// TIA Portal project "ManufacturingCell2_ATOLE" (V19)

(* hardware
DEVICE "S7-1200 station_1"  S7-1200 Station
   slot 0: "Rack_0"  S7-1200 Rack  Rack  V1.0
   slot 1: "PLC_Machining"  CPU 1214C AC/DC/Rly  6ES7 214-1BG40-0XB0  V4.5
   slot 2: "DI 16x24VDC/DQ 16xRelay_1"  SM 1223 DI16/DQ16 x relay  6ES7 223-1PL32-0XB0  V2.0
   slot 3: "AQ 1x12BIT_1"  AQ1 signal board  6ES7 232-4HA30-0XB0  V1.0
   slot 3: "AI 4x13BIT/AQ 2x14BIT_1"  6ES7 234-4HE32-0XB0  V2.1
DEVICE "Machining_HMI"  KTP700 Basic PN
   slot 0: "HMI_1"  KTP700 Basic PN  6AV2 123-2GB03-0AX0  17.0.0.0
   slot 1: "HMI_RT_1"  KTP700 Basic PN  6AV2 123-2GB03-0AX0  17.0.0.0
   slot 5: "HMI_1.IE_CP_1"  PROFINET Interface  17.0.0.0
      slot 1: "PROFINET Interface_1"  PROFINET Interface
         slot 1: "Port_1"  Port
DEVICE "S7-1200 station_2"  S7-1200 Station
   slot 0: "Rack_0"  S7-1200 Rack  Rack  V1.0
   slot 1: "PLC_Pneumatic"  CPU 1214C AC/DC/Rly  6ES7 214-1BG40-0XB0  V4.5
   slot 2: "DI 16x24VDC/DQ 16xRelay_1"  SM 1223 DI16/DQ16 x relay  6ES7 223-1PL32-0XB0  V2.0
   slot 3: "AQ 1x12BIT_1"  AQ1 signal board  6ES7 232-4HA30-0XB0  V1.0
   slot 3: "AI 4x13BIT/AQ 2x14BIT_1"  6ES7 234-4HE32-0XB0  V2.1
DEVICE "Pneumatic_HMI"  KTP700 Basic PN
   slot 0: "HMI_2"  KTP700 Basic PN  6AV2 123-2GB03-0AX0  17.0.0.0
   slot 1: "HMI_RT_2"  KTP700 Basic PN  6AV2 123-2GB03-0AX0  17.0.0.0
   slot 5: "HMI_2.IE_CP_1"  PROFINET Interface  17.0.0.0
      slot 1: "PROFINET Interface_1"  PROFINET Interface
         slot 1: "Port_1"  Port
*)

// ===== PLC "PLC_Machining"  CPU 1214C AC/DC/Rly =====

VAR_GLOBAL   // PLC tag table "Default tag table"
   "Pusher_latch" AT %M10.0 : Bool;
   "Conveyor2_latch" AT %M10.1 : Bool;
   "Conveyor4_latch" AT %M10.2 : Bool;
   "Conveyor3_latch" AT %M10.3 : Bool;
   "Conveyor5_latch" AT %M10.4 : Bool;
   "Conveyor6_IN_latch" AT %M10.5 : Bool;
   "Conveyor6_OUT_latch" AT %M10.6 : Bool;
   "Conveyor6_Position" AT %M10.7 : Bool;
   "lampBlinkTag" AT %M11.0 : Bool;
   "cakeFlavor" AT %MW12 : UInt;
   "drillingTime" AT %MD14 : Time;
   "mixingTime" AT %MD18 : Time;
   "System_Byte" AT %MB22 : Byte;
   "FirstScan" AT %M22.0 : Bool;
   "DiagStatusUpdate" AT %M22.1 : Bool;
   "AlwaysTRUE" AT %M22.2 : Bool;
   "AlwaysFALSE" AT %M22.3 : Bool;
   "drillActive" AT %M23.0 : Bool;
   "mixActive" AT %M23.1 : Bool;
   "CognexID" AT %MW24 : Int;
   "manualModeSW_memory" AT %M23.2 : Bool;
   "CognexID_UInt" AT %MW26 : UInt;
   "SetCognexID_Edge" AT %M23.3 : Bool;
   "OptoDrill_Edge" AT %M23.4 : Bool;
   "OptoMix_Edge" AT %M23.5 : Bool;
   "Power_consumption" AT %MD28 : Real;
   "Conveyor6_OUT_Finish" AT %M11.1 : Bool;
   "Conveyor6Finish_TP_Edge" AT %M11.2 : Bool;
END_VAR

VAR_GLOBAL   // PLC tag table "M_HMI_Tags"
   "HMI_BTN_Conveyor2" AT %M50.1 : Bool;
   "HMI_BTN_Pusher1" AT %M50.2 : Bool;
   "HMI_BTN_Conveyor3" AT %M50.3 : Bool;
   "HMI_BTN_Conveyor4" AT %M50.4 : Bool;
   "HMI_BTN_Conveyor5" AT %M50.5 : Bool;
   "HMI_BTN_Drill" AT %M50.6 : Bool;
   "HMI_BTN_Mix" AT %M50.7 : Bool;
   "HMI_BTN1" AT %M50.0 : Bool;
   "HMI_BTN_Pusher2" AT %M51.0 : Bool;
   "HMI_BTN_Conveyor6IN" AT %M51.1 : Bool;
   "HMI_BTN_Conveyor6OUT" AT %M51.2 : Bool;
   "HMI_BTN_PressDown" AT %M51.3 : Bool;
   "HMI_BTN_PressUp" AT %M51.4 : Bool;
   "HMI_BTN_PlantView" AT %M51.5 : Bool;
   "HMI_BTN_ProcessTimes" AT %M51.6 : Bool;
   "HMI_BTN_ManualControl" AT %M51.7 : Bool;
   "HMI_BTN17" AT %M52.0 : Bool;
   "HMI_BTN18" AT %M52.1 : Bool;
   "HMI_BTN19" AT %M52.2 : Bool;
   "HMI_BTN20" AT %M52.3 : Bool;
   "HMI_BTN21" AT %M52.4 : Bool;
   "HMI_BTN22" AT %M52.5 : Bool;
   "HMI_BTN23" AT %M52.6 : Bool;
   "HMI_BTN24" AT %M52.7 : Bool;
   "ManualMode_SW" AT %M53.0 : Bool;
   "HMI_SetScreen" AT %MW54 : Int;
END_VAR

VAR_GLOBAL   // PLC tag table "M_Cell_Tags"
   "Opto_Conveyor2A" AT %I0.0 : Bool;
   "Opto_Conveyor2B" AT %I0.1 : Bool;
   "Green_BTN" AT %I9.4 : Bool;
   "Yellow_BTN" AT %I9.5 : Bool;
   "Red_BTN" AT %I9.6 : Bool;
   "Emergency_BTN" AT %I9.7 : Bool;
   "Pusher1_BTN" AT %I0.2 : Bool;
   "Opto_Drill" AT %I0.3 : Bool;
   "Opto_Mix" AT %I0.4 : Bool;
   "Opto_Conveyor5" AT %I0.6 : Bool;
   "Pusher2_BTN" AT %I0.5 : Bool;
   "Opto_Conveyor6A" AT %I8.1 : Bool;
   "Opto_Conveyor6B" AT %I8.0 : Bool;
   "Press_BTN_DOWN" AT %I8.2 : Bool;
   "Press_BTN_UP" AT %I8.3 : Bool;
   "Conveyor2_tactileSW" AT %I0.7 : Bool;
   "cellPotentiometer" AT %IW64 : Int;
   "Cognex_out0" AT %I9.0 : Bool;
   "Cognex_out1" AT %I9.1 : Bool;
   "Cognex_out2" AT %I9.2 : Bool;
   "Green_Light" AT %Q9.5 : Bool;
   "Red_Light" AT %Q9.6 : Bool;
   "Blue_Light" AT %Q9.7 : Bool;
   "Conveyor2" AT %Q0.0 : Bool;
   "Pusher1" AT %Q0.1 : Bool;
   "Conveyor4" AT %Q0.4 : Bool;
   "Conveyor5" AT %Q0.7 : Bool;
   "Conveyor3" AT %Q0.2 : Bool;
   "Drill" AT %Q0.3 : Bool;
   "Mix" AT %Q0.5 : Bool;
   "Pusher2" AT %Q0.6 : Bool;
   "Green_Tower" AT %Q1.0 : Bool;
   "Red_Tower" AT %Q1.1 : Bool;
   "Conveyor6_OUT" AT %Q8.3 : Bool;
   "Press_UP" AT %Q8.4 : Bool;
   "Press_DOWN" AT %Q8.5 : Bool;
   "Conveyor6_IN" AT %Q8.2 : Bool;
   "AO_Channel0" AT %QW112 : Int;
   "AO_Channel1" AT %QW114 : Int;
   "AO_Cell" AT %QW80 : Int;
   "Cognex_in0" AT %Q8.7 : Bool;
END_VAR

VAR_GLOBAL   // PLC tag table "Clock_Tags"
   "Clock_Byte" AT %MB0 : Byte;
   "Clock_10Hz" AT %M0.0 : Bool;
   "Clock_5Hz" AT %M0.1 : Bool;
   "Clock_2.5Hz" AT %M0.2 : Bool;
   "Clock_2Hz" AT %M0.3 : Bool;
   "Clock_1.25Hz" AT %M0.4 : Bool;
   "Clock_1Hz" AT %M0.5 : Bool;
   "Clock_0.625Hz" AT %M0.6 : Bool;
   "Clock_0.5Hz" AT %M0.7 : Bool;
END_VAR

DATA_BLOCK "potentiometerValue"   // DB14
{ S7_Optimized_Access := 'TRUE' }
VERSION : 0.1
// stored: InstanceOfName FB_AnalogInput
"FB_AnalogInput"
BEGIN
END_DATA_BLOCK

DATA_BLOCK "processTimes_DB"   // DB15
{ S7_Optimized_Access := 'TRUE' }
VERSION : 0.1
   VAR
      chocolateDrillingInput_ms : UInt := 6000;
      chocolateMixingInput_ms : UInt := 6000;
      vanillaDrillingInput_ms : UInt := 7000;
      vanillaMixingInput_ms : UInt := 7000;
      strawberryDrillingInput_ms : UInt := 8000;
      strawberryMixingInput_ms : UInt := 8000;
      chocolateDrilling_s : Time;
      chocolateMixing_s : Time;
      vanillaDrilling_s : Time;
      vanillaMixing_s : Time;
      strawberryDrilling_s : Time;
      strawberryMixing_s : Time;
   END_VAR
BEGIN
END_DATA_BLOCK

DATA_BLOCK "Mix_FIFO_DB"   // DB18
{ S7_Optimized_Access := 'TRUE' }
VERSION : 0.1
   VAR
      "Array" : Array[0..99] of Int;
      Index : Int;
      ServiceIndex : Int;
      ServiceIndex_UInt : UInt;
   END_VAR
BEGIN
END_DATA_BLOCK

DATA_BLOCK "Drill_FIFO_DB"   // DB19
{ S7_Optimized_Access := 'TRUE' }
VERSION : 0.1
   VAR
      "Array" : Array[0..99] of Int;
      Index : Int;
      ServiceIndex : Int;
      ServiceIndex_UInt : UInt;
   END_VAR
BEGIN
END_DATA_BLOCK

DATA_BLOCK "Cobot_FIFO_DB"   // DB20
{ S7_Optimized_Access := 'TRUE' }
VERSION : 0.1
   VAR
      "Array" : Array[0..99] of Int;
      Index : Int;
      ServiceIndex : Int;
      ServiceIndex_UInt : UInt;
   END_VAR
BEGIN
END_DATA_BLOCK

DATA_BLOCK "Python_Gateway_DB"   // DB99
{ S7_Optimized_Access := 'FALSE' }
VERSION : 0.1
   VAR
      emergencyStop_Pneumatic : Bool;
      emergencyStop_Machining : Bool;
      cobotIsMoving : Bool;
      PneumaticPower : Real;
      MachiningPower : Real;
      AirPressure : Real;
      ChocolateUnitsFinished : Int;
      VanillaUnitsFinished : Int;
      StrawberryUnitsFinished : Int;
      OnlineUser : String[40];
      OnlineRole : String[30];
      CognexID : Int;
   END_VAR
BEGIN
END_DATA_BLOCK

DATA_BLOCK "Machining_Communication_DB"   // DB100
{ S7_Optimized_Access := 'FALSE' }
VERSION : 0.1
   VAR
      Cognex_Code : Int;   // Machining to Pneu
      Conveyor5_Done : Bool;   // Machining to Pneu
      Conveyor2_SensorA : Bool;   // Machining to Pneu
      ShutterTP_Q : Bool;   // Machining to Pneu
      Conveyor6Out_Finish : Bool;   // Machining to Pneu
      CobotCode_Palletizing : Byte;   // Machining to Pneu
      ReadCobotCode : Byte;   // Pneu to Machining
      Cognex_Shutter : Bool;   // Pneu to Machining
      Conveyor1_Sensor : Bool;   // Pneu to Machining
      Cobot_Moving : Bool;   // Pneu to Machining
      Pneumatic_EmergencyBTN : Bool;   // Pneu to Machining
      SetCognexID : Bool;   // Pneu to Machining
      M_PlantView : Bool;   // Pneu to Machining
      M_ManualControl : Bool;   // Pneu to Machining
      M_ProcessTimes : Bool;   // Pneu to Machining
      HMI_BTN_Enter : Bool;   // Pneu to Machining
      HMI_BTN_Logout : Bool;   // Pneu to Machining
      PneumaticPower : Real;   // Pneu to Machining
      AirPressure : Real;   // Pneu to Machining
      ActiveUser : String[40];   // Pneu to Machining
      ActiveRole : String[30];   // Pneu to Machining
      ChocolateCount : Int;   // Pneu to Machining
      VanillaCount : Int;   // Pneu to Machining
      StrawberryCount : Int;   // Pneu to Machining
   END_VAR
BEGIN
END_DATA_BLOCK

// folder: System blocks/Program resources

DATA_BLOCK "Mix_PostTP"   // DB1
{ S7_Optimized_Access := 'TRUE' }
AUTHOR : Simatic
FAMILY : IEC
NAME : IEC_TMR
VERSION : 1.0
// stored: InstanceOfName IEC_TIMER
"IEC_TIMER"
BEGIN
END_DATA_BLOCK

DATA_BLOCK "Pusher1_Delay"   // DB2
{ S7_Optimized_Access := 'TRUE' }
AUTHOR : Simatic
FAMILY : IEC
NAME : IEC_TMR
VERSION : 1.0
// stored: InstanceOfName IEC_TIMER
"IEC_TIMER"
BEGIN
END_DATA_BLOCK

DATA_BLOCK "Drill_OperationTP"   // DB3
{ S7_Optimized_Access := 'TRUE' }
AUTHOR : Simatic
FAMILY : IEC
NAME : IEC_TMR
VERSION : 1.0
// stored: InstanceOfName IEC_TIMER
"IEC_TIMER"
BEGIN
END_DATA_BLOCK

DATA_BLOCK "Mix_OperationTP"   // DB4
{ S7_Optimized_Access := 'TRUE' }
AUTHOR : Simatic
FAMILY : IEC
NAME : IEC_TMR
VERSION : 1.0
// stored: InstanceOfName IEC_TIMER
"IEC_TIMER"
BEGIN
END_DATA_BLOCK

DATA_BLOCK "Drill_PostTP"   // DB5
{ S7_Optimized_Access := 'TRUE' }
AUTHOR : Simatic
FAMILY : IEC
NAME : IEC_TMR
VERSION : 1.0
// stored: InstanceOfName IEC_TIMER
"IEC_TIMER"
BEGIN
END_DATA_BLOCK

DATA_BLOCK "Conveyor2_TP"   // DB6
{ S7_Optimized_Access := 'TRUE' }
AUTHOR : Simatic
FAMILY : IEC
NAME : IEC_TMR
VERSION : 1.0
// stored: InstanceOfName IEC_TIMER
"IEC_TIMER"
BEGIN
END_DATA_BLOCK

DATA_BLOCK "Conveyor2_ManualDelay"   // DB7
{ S7_Optimized_Access := 'TRUE' }
AUTHOR : Simatic
FAMILY : IEC
NAME : IEC_TMR
VERSION : 1.0
// stored: InstanceOfName IEC_TIMER
"IEC_TIMER"
BEGIN
END_DATA_BLOCK

DATA_BLOCK "Pusher2_Delay"   // DB8
{ S7_Optimized_Access := 'TRUE' }
AUTHOR : Simatic
FAMILY : IEC
NAME : IEC_TMR
VERSION : 1.0
// stored: InstanceOfName IEC_TIMER
"IEC_TIMER"
BEGIN
END_DATA_BLOCK

DATA_BLOCK "Press_Delay"   // DB9
{ S7_Optimized_Access := 'TRUE' }
AUTHOR : Simatic
FAMILY : IEC
NAME : IEC_TMR
VERSION : 1.0
// stored: InstanceOfName IEC_TIMER
"IEC_TIMER"
BEGIN
END_DATA_BLOCK

DATA_BLOCK "IEC_Timer_0_DB"   // DB10
{ S7_Optimized_Access := 'TRUE' }
AUTHOR : Simatic
FAMILY : IEC
NAME : IEC_TMR
VERSION : 1.0
// stored: InstanceOfName IEC_TIMER
"IEC_TIMER"
BEGIN
END_DATA_BLOCK

DATA_BLOCK "Press_DOWN_Timer"   // DB11
{ S7_Optimized_Access := 'TRUE' }
AUTHOR : Simatic
FAMILY : IEC
NAME : IEC_TMR
VERSION : 1.0
// stored: InstanceOfName IEC_TIMER
"IEC_TIMER"
BEGIN
END_DATA_BLOCK

DATA_BLOCK "Emergency_Blink_TP"   // DB12
{ S7_Optimized_Access := 'TRUE' }
AUTHOR : Simatic
FAMILY : IEC
NAME : IEC_TMR
VERSION : 1.0
// stored: InstanceOfName IEC_TIMER
"IEC_TIMER"
BEGIN
END_DATA_BLOCK

DATA_BLOCK "Emergency_Blink_TON"   // DB13
{ S7_Optimized_Access := 'TRUE' }
AUTHOR : Simatic
FAMILY : IEC
NAME : IEC_TMR
VERSION : 1.0
// stored: InstanceOfName IEC_TIMER
"IEC_TIMER"
BEGIN
END_DATA_BLOCK

DATA_BLOCK "Shutter_TP"   // DB16
{ S7_Optimized_Access := 'TRUE' }
AUTHOR : Simatic
FAMILY : IEC
NAME : IEC_TMR
VERSION : 1.0
// stored: InstanceOfName IEC_TIMER
"IEC_TIMER"
BEGIN
END_DATA_BLOCK

DATA_BLOCK "startupDelay_TP"   // DB17
{ S7_Optimized_Access := 'TRUE' }
AUTHOR : Simatic
FAMILY : IEC
NAME : IEC_TMR
VERSION : 1.0
// stored: InstanceOfName IEC_TIMER
"IEC_TIMER"
BEGIN
END_DATA_BLOCK

DATA_BLOCK "conveyor6Transmit_TP"   // DB21
{ S7_Optimized_Access := 'TRUE' }
AUTHOR : Simatic
FAMILY : IEC
NAME : IEC_TMR
VERSION : 1.0
// stored: InstanceOfName IEC_TIMER
"IEC_TIMER"
BEGIN
END_DATA_BLOCK

DATA_BLOCK "ConveyorCobotByte_TON"   // DB22
{ S7_Optimized_Access := 'TRUE' }
AUTHOR : Simatic
FAMILY : IEC
NAME : IEC_TMR
VERSION : 1.0
// stored: InstanceOfName IEC_TIMER
"IEC_TIMER"
BEGIN
END_DATA_BLOCK

DATA_BLOCK "Conveyor6Finish_TP"   // DB23
{ S7_Optimized_Access := 'TRUE' }
AUTHOR : Simatic
FAMILY : IEC
NAME : IEC_TMR
VERSION : 1.0
// stored: InstanceOfName IEC_TIMER
"IEC_TIMER"
BEGIN
END_DATA_BLOCK

DATA_BLOCK "SendCognexCodePy_TON"   // DB24
{ S7_Optimized_Access := 'TRUE' }
AUTHOR : Simatic
FAMILY : IEC
NAME : IEC_TMR
VERSION : 1.0
// stored: InstanceOfName IEC_TIMER
"IEC_TIMER"
BEGIN
END_DATA_BLOCK

// folder: (top level)

FUNCTION_BLOCK "FB_AnalogInput"   // FB1, LAD
{ S7_Optimized_Access := 'TRUE' }
VERSION : 0.1
   VAR_INPUT
      minRaw : Int;
      maxRaw : Int := 27648;
      rawValue : Int;
      minScale : Real;
      maxScale : Real := 1.0;
   END_VAR
   VAR_OUTPUT
      outputValue : Real;
   END_VAR
   VAR_TEMP
      normValue : Real;
   END_VAR
BEGIN

REGION Network 1
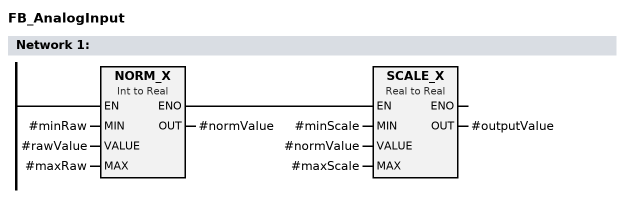
   RUNG wire#powerrail
      { S7_Templates := "[SrcType := Int, DestType := Real]" } Normalize(min := #minRaw, value := #rawValue, max := #maxRaw, out => #normValue)
      { S7_Templates := "[SrcType := Real, DestType := Real]" } Scale(min := #minScale, value := #normValue, max := #maxScale, out => #outputValue)
   END_RUNG
   // the same network as SCL:
   #normValue := NORM_X(MIN := #minRaw, VALUE := #rawValue, MAX := #maxRaw);
   #outputValue := SCALE_X(MIN := #minScale, VALUE := #normValue, MAX := #maxScale);
END_REGION
END_FUNCTION_BLOCK

ORGANIZATION_BLOCK "Main_Machining"   // OB1, LAD, ProgramCycle
{ S7_Optimized_Access := 'TRUE' }
VERSION : 0.1
   VAR_INPUT
      Initial_Call : Bool;
      Remanence : Bool;
   END_VAR
   VAR_TEMP   // added for the SCL form of the ladder/FBD networks
      _w1 : Bool;
      _w2 : Bool;
   END_VAR
BEGIN

REGION Network 1: Startup Delay
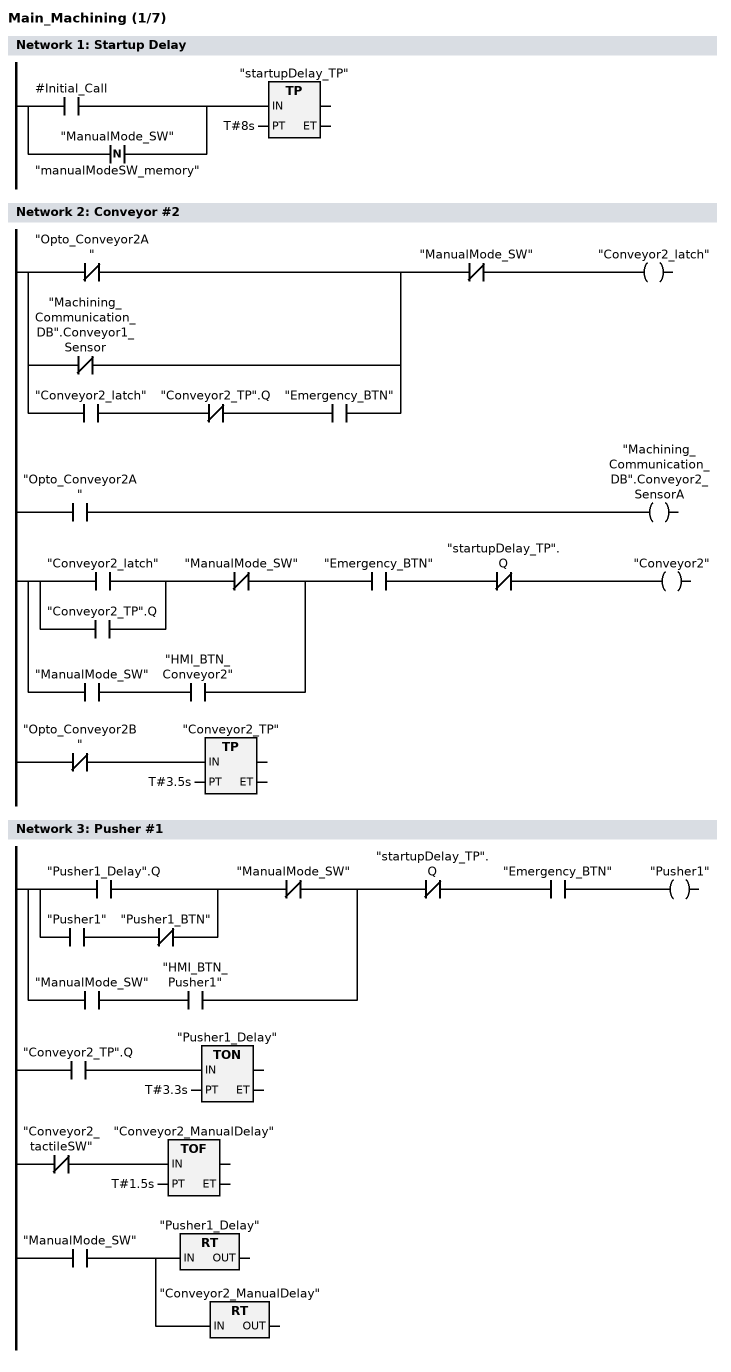
   #_w1 := NOT "ManualMode_SW" AND "manualModeSW_memory";   // falling edge of "ManualMode_SW"
   "manualModeSW_memory" := "ManualMode_SW";
   "startupDelay_TP".TP(IN := #Initial_Call OR #_w1, PT := T#8s);
END_REGION

REGION Network 2: Conveyor #2
   "Conveyor2_latch" := (NOT "Opto_Conveyor2A" OR NOT "Machining_Communication_DB".Conveyor1_Sensor OR ("Conveyor2_latch" AND NOT "Conveyor2_TP".Q AND "Emergency_BTN")) AND NOT "ManualMode_SW";
   "Machining_Communication_DB".Conveyor2_SensorA := "Opto_Conveyor2A";
   "Conveyor2" := ((("Conveyor2_latch" OR "Conveyor2_TP".Q) AND NOT "ManualMode_SW") OR ("ManualMode_SW" AND "HMI_BTN_Conveyor2")) AND "Emergency_BTN" AND NOT "startupDelay_TP".Q;
   "Conveyor2_TP".TP(IN := NOT "Opto_Conveyor2B", PT := T#3.5s);
END_REGION

REGION Network 3: Pusher #1
   "Pusher1" := ((("Pusher1_Delay".Q OR ("Pusher1" AND NOT "Pusher1_BTN")) AND NOT "ManualMode_SW") OR ("ManualMode_SW" AND "HMI_BTN_Pusher1")) AND NOT "startupDelay_TP".Q AND "Emergency_BTN";
   "Pusher1_Delay".TON(IN := "Conveyor2_TP".Q, PT := T#3.3s);
   "Conveyor2_ManualDelay".TOF(IN := NOT "Conveyor2_tactileSW", PT := T#1.5s);
   IF "ManualMode_SW" THEN
       RESET_TIMER("Pusher1_Delay");
       RESET_TIMER("Conveyor2_ManualDelay");
   END_IF;
END_REGION

REGION Network 4: Conveyor #3
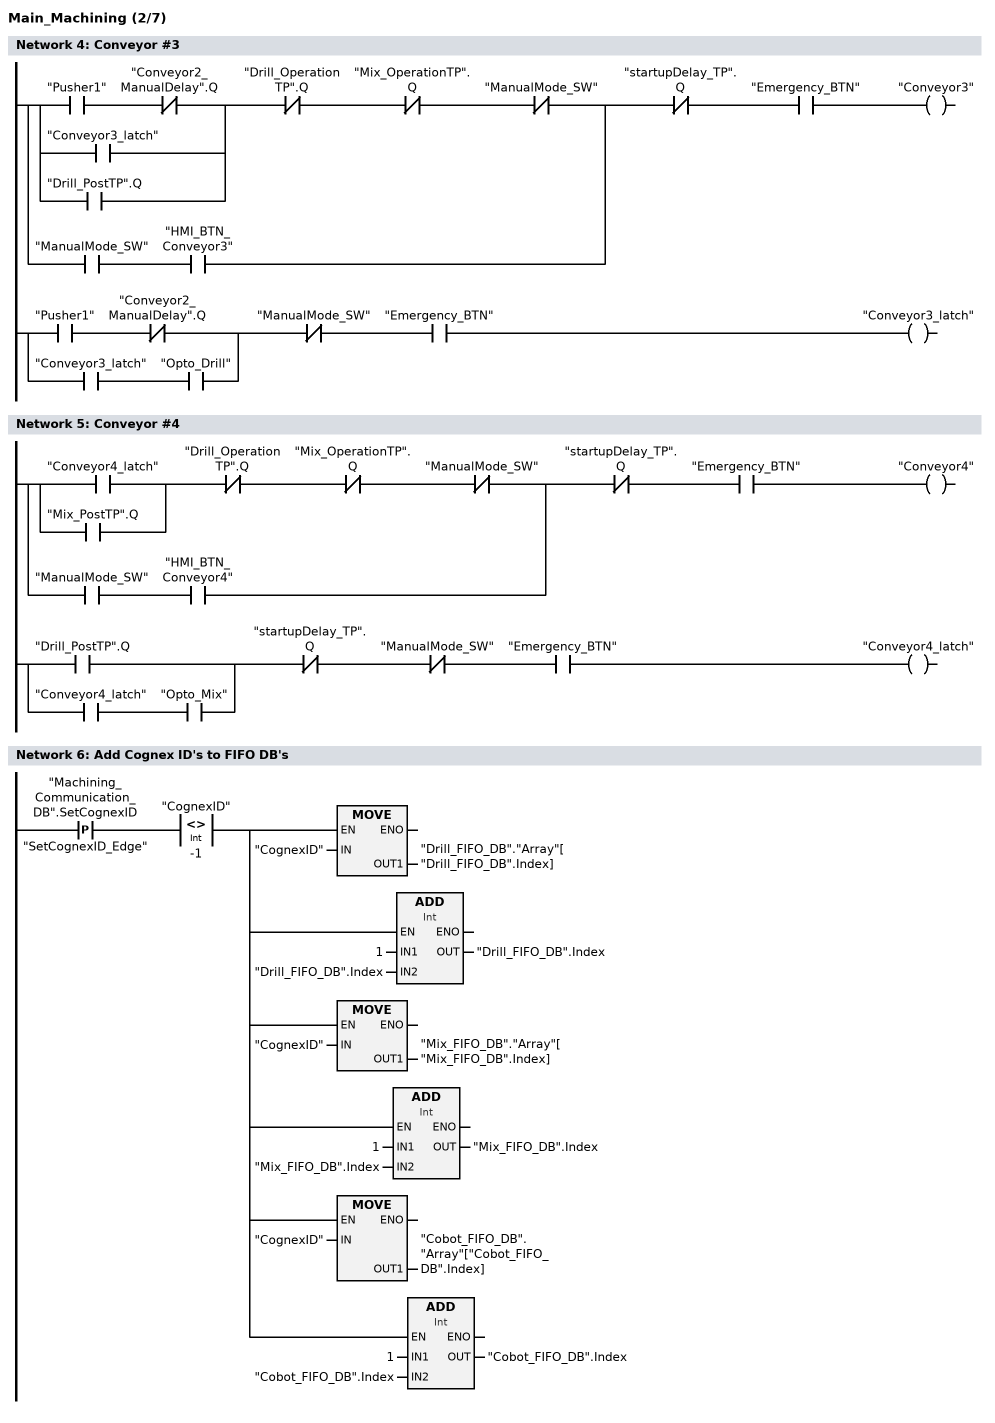
   RUNG wire#powerrail
      Contact( "Pusher1" )
      I_Contact( "Conveyor2_ManualDelay".Q )
      wire#w1
      I_Contact( "Drill_OperationTP".Q )
      I_Contact( "Mix_OperationTP".Q )
      I_Contact( "ManualMode_SW" )
      wire#w2
      I_Contact( "startupDelay_TP".Q )
      Contact( "Emergency_BTN" )
      Coil( "Conveyor3" )
   END_RUNG
   RUNG wire#powerrail
      Contact( "Conveyor3_latch" )
   END_RUNG wire#w1
   RUNG wire#powerrail
      Contact( "Drill_PostTP".Q )
   END_RUNG wire#w1
   RUNG wire#powerrail
      Contact( "ManualMode_SW" )
      Contact( "HMI_BTN_Conveyor3" )
   END_RUNG wire#w2
   RUNG wire#powerrail
      Contact( "Pusher1" )
      I_Contact( "Conveyor2_ManualDelay".Q )
      wire#w3
      I_Contact( "ManualMode_SW" )
      Contact( "Emergency_BTN" )
      Coil( "Conveyor3_latch" )
   END_RUNG
   RUNG wire#powerrail
      Contact( "Conveyor3_latch" )
      Contact( "Opto_Drill" )
   END_RUNG wire#w3
   // the same network as SCL:
   "Conveyor3" := (((("Pusher1" AND NOT "Conveyor2_ManualDelay".Q) OR "Conveyor3_latch" OR "Drill_PostTP".Q) AND NOT "Drill_OperationTP".Q AND NOT "Mix_OperationTP".Q AND NOT "ManualMode_SW") OR ("ManualMode_SW" AND "HMI_BTN_Conveyor3")) AND NOT "startupDelay_TP".Q AND "Emergency_BTN";
   "Conveyor3_latch" := (("Pusher1" AND NOT "Conveyor2_ManualDelay".Q) OR ("Conveyor3_latch" AND "Opto_Drill")) AND NOT "ManualMode_SW" AND "Emergency_BTN";
END_REGION

REGION Network 5: Conveyor #4
   RUNG wire#powerrail
      Contact( "Conveyor4_latch" )
      wire#w1
      I_Contact( "Drill_OperationTP".Q )
      I_Contact( "Mix_OperationTP".Q )
      I_Contact( "ManualMode_SW" )
      wire#w2
      I_Contact( "startupDelay_TP".Q )
      Contact( "Emergency_BTN" )
      Coil( "Conveyor4" )
   END_RUNG
   RUNG wire#powerrail
      Contact( "Mix_PostTP".Q )
   END_RUNG wire#w1
   RUNG wire#powerrail
      Contact( "ManualMode_SW" )
      Contact( "HMI_BTN_Conveyor4" )
   END_RUNG wire#w2
   RUNG wire#powerrail
      Contact( "Drill_PostTP".Q )
      wire#w3
      I_Contact( "startupDelay_TP".Q )
      I_Contact( "ManualMode_SW" )
      Contact( "Emergency_BTN" )
      Coil( "Conveyor4_latch" )
   END_RUNG
   RUNG wire#powerrail
      Contact( "Conveyor4_latch" )
      Contact( "Opto_Mix" )
   END_RUNG wire#w3
   // the same network as SCL:
   "Conveyor4" := ((("Conveyor4_latch" OR "Mix_PostTP".Q) AND NOT "Drill_OperationTP".Q AND NOT "Mix_OperationTP".Q AND NOT "ManualMode_SW") OR ("ManualMode_SW" AND "HMI_BTN_Conveyor4")) AND NOT "startupDelay_TP".Q AND "Emergency_BTN";
   "Conveyor4_latch" := ("Drill_PostTP".Q OR ("Conveyor4_latch" AND "Opto_Mix")) AND NOT "startupDelay_TP".Q AND NOT "ManualMode_SW" AND "Emergency_BTN";
END_REGION

REGION Network 6: Add Cognex ID's to FIFO DB's
   RUNG wire#powerrail
      P_Contact(operand := "Machining_Communication_DB".SetCognexID, bit := "SetCognexID_Edge")
      { S7_Templates := "SrcType := Int" } NE_Contact(in1 := "CognexID", in2 := -1)
      wire#w1
      Move(in := "CognexID", out1 => "Drill_FIFO_DB"."Array"["Drill_FIFO_DB".Index])
   END_RUNG
   RUNG wire#w1
      { S7_Templates := "SrcType := Int" } Add(in1 := 1, in2 := "Drill_FIFO_DB".Index, out => "Drill_FIFO_DB".Index)
   END_RUNG
   RUNG wire#w1
      Move(in := "CognexID", out1 => "Mix_FIFO_DB"."Array"["Mix_FIFO_DB".Index])
   END_RUNG
   RUNG wire#w1
      { S7_Templates := "SrcType := Int" } Add(in1 := 1, in2 := "Mix_FIFO_DB".Index, out => "Mix_FIFO_DB".Index)
   END_RUNG
   RUNG wire#w1
      Move(in := "CognexID", out1 => "Cobot_FIFO_DB"."Array"["Cobot_FIFO_DB".Index])
   END_RUNG
   RUNG wire#w1
      { S7_Templates := "SrcType := Int" } Add(in1 := 1, in2 := "Cobot_FIFO_DB".Index, out => "Cobot_FIFO_DB".Index)
   END_RUNG
   // the same network as SCL:
   #_w1 := "Machining_Communication_DB".SetCognexID AND NOT "SetCognexID_Edge";   // rising edge of "Machining_Communication_DB".SetCognexID
   "SetCognexID_Edge" := "Machining_Communication_DB".SetCognexID;
   IF #_w1 AND ("CognexID" <> (-1)) THEN
       "Drill_FIFO_DB"."Array"["Drill_FIFO_DB".Index] := "CognexID";
       "Drill_FIFO_DB".Index := 1 + "Drill_FIFO_DB".Index;
       "Mix_FIFO_DB"."Array"["Mix_FIFO_DB".Index] := "CognexID";
       "Mix_FIFO_DB".Index := 1 + "Mix_FIFO_DB".Index;
       "Cobot_FIFO_DB"."Array"["Cobot_FIFO_DB".Index] := "CognexID";
       "Cobot_FIFO_DB".Index := 1 + "Cobot_FIFO_DB".Index;
   END_IF;
END_REGION

REGION Network 7: Set drilling and mixing times
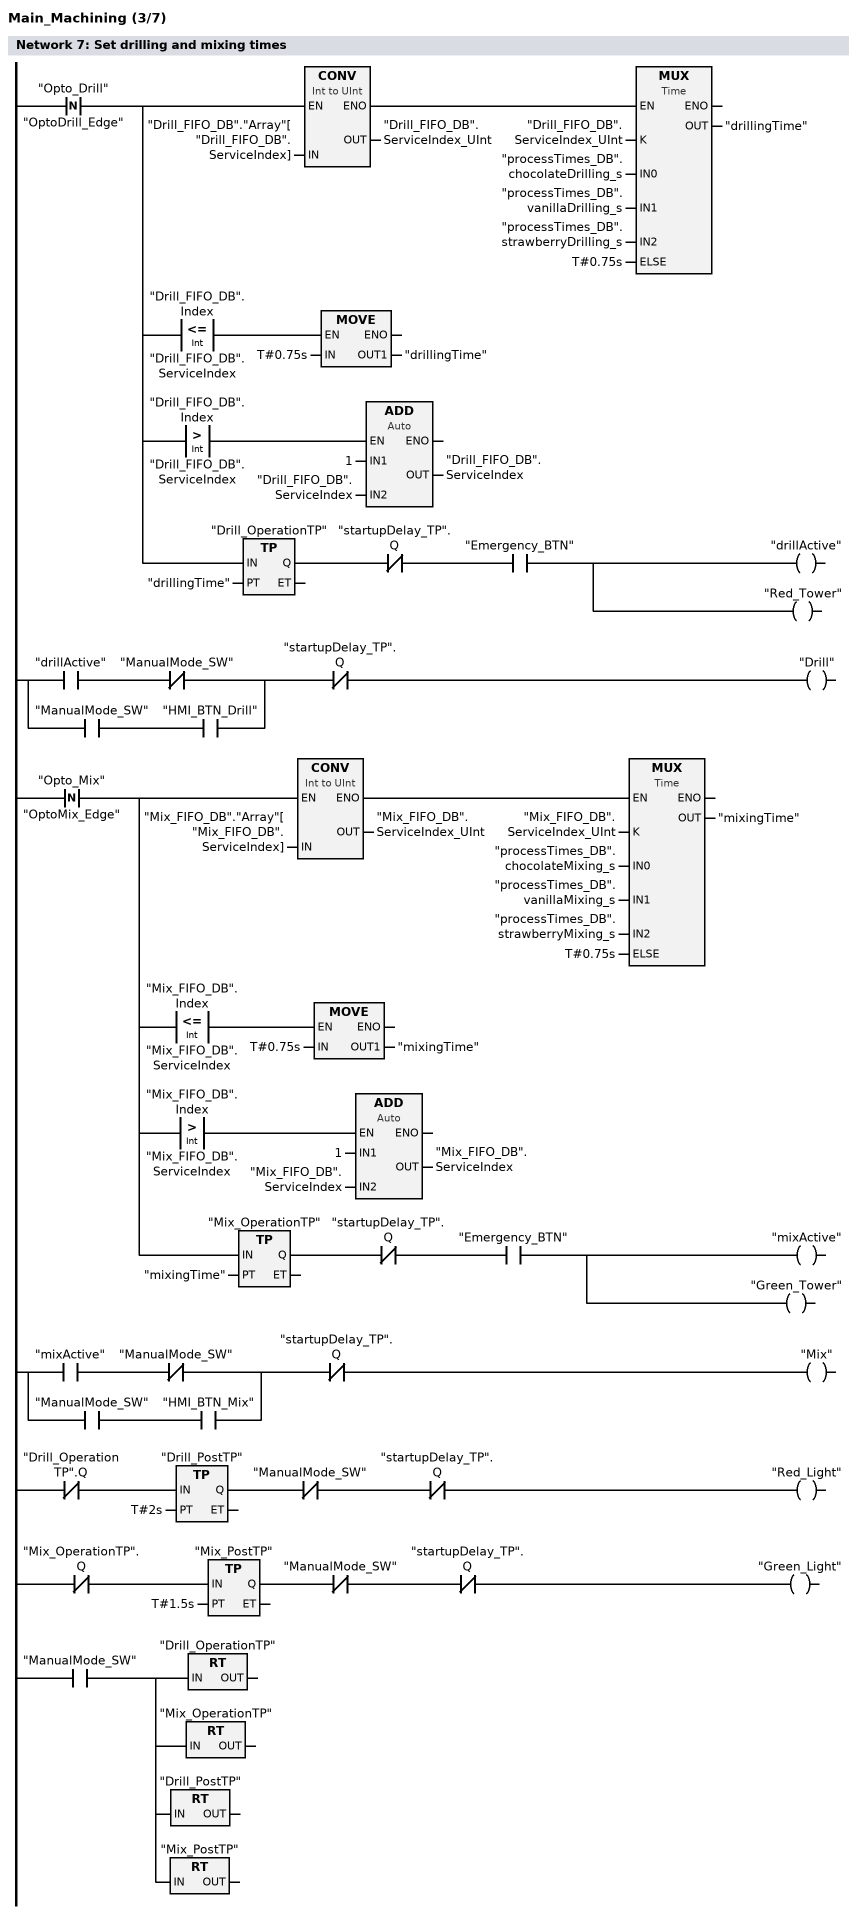
   // no SCL statement known for Mux: written as a call
   #_w1 := NOT "Opto_Drill" AND "OptoDrill_Edge";   // falling edge of "Opto_Drill"
   "OptoDrill_Edge" := "Opto_Drill";
   IF #_w1 THEN
       "Drill_FIFO_DB".ServiceIndex_UInt := INT_TO_UINT("Drill_FIFO_DB"."Array"["Drill_FIFO_DB".ServiceIndex]);
       Mux(k := "Drill_FIFO_DB".ServiceIndex_UInt,
           in0 := "processTimes_DB".chocolateDrilling_s,
           in1 := "processTimes_DB".vanillaDrilling_s,
           in2 := "processTimes_DB".strawberryDrilling_s,
           "else" := T#0.75s,
           out => "drillingTime");
   END_IF;
   IF #_w1 AND ("Drill_FIFO_DB".Index <= "Drill_FIFO_DB".ServiceIndex) THEN
       "drillingTime" := T#0.75s;
   END_IF;
   IF #_w1 AND ("Drill_FIFO_DB".Index > "Drill_FIFO_DB".ServiceIndex) THEN
       "Drill_FIFO_DB".ServiceIndex := 1 + "Drill_FIFO_DB".ServiceIndex;
   END_IF;
   "Drill_OperationTP".TP(IN := #_w1, PT := "drillingTime");
   "drillActive" := "Drill_OperationTP".Q AND NOT "startupDelay_TP".Q AND "Emergency_BTN";
   "Red_Tower" := "drillActive";
   "Drill" := (("drillActive" AND NOT "ManualMode_SW") OR ("ManualMode_SW" AND "HMI_BTN_Drill")) AND NOT "startupDelay_TP".Q;
   #_w2 := NOT "Opto_Mix" AND "OptoMix_Edge";   // falling edge of "Opto_Mix"
   "OptoMix_Edge" := "Opto_Mix";
   IF #_w2 THEN
       "Mix_FIFO_DB".ServiceIndex_UInt := INT_TO_UINT("Mix_FIFO_DB"."Array"["Mix_FIFO_DB".ServiceIndex]);
       Mux(k := "Mix_FIFO_DB".ServiceIndex_UInt,
           in0 := "processTimes_DB".chocolateMixing_s,
           in1 := "processTimes_DB".vanillaMixing_s,
           in2 := "processTimes_DB".strawberryMixing_s,
           "else" := T#0.75s,
           out => "mixingTime");
   END_IF;
   IF #_w2 AND ("Mix_FIFO_DB".Index <= "Mix_FIFO_DB".ServiceIndex) THEN "mixingTime" := T#0.75s; END_IF;
   IF #_w2 AND ("Mix_FIFO_DB".Index > "Mix_FIFO_DB".ServiceIndex) THEN
       "Mix_FIFO_DB".ServiceIndex := 1 + "Mix_FIFO_DB".ServiceIndex;
   END_IF;
   "Mix_OperationTP".TP(IN := #_w2, PT := "mixingTime");
   "mixActive" := "Mix_OperationTP".Q AND NOT "startupDelay_TP".Q AND "Emergency_BTN";
   "Green_Tower" := "mixActive";
   "Mix" := (("mixActive" AND NOT "ManualMode_SW") OR ("ManualMode_SW" AND "HMI_BTN_Mix")) AND NOT "startupDelay_TP".Q;
   "Drill_PostTP".TP(IN := NOT "Drill_OperationTP".Q, PT := T#2s);
   "Red_Light" := "Drill_PostTP".Q AND NOT "ManualMode_SW" AND NOT "startupDelay_TP".Q;
   "Mix_PostTP".TP(IN := NOT "Mix_OperationTP".Q, PT := T#1.5s);
   "Green_Light" := "Mix_PostTP".Q AND NOT "ManualMode_SW" AND NOT "startupDelay_TP".Q;
   IF "ManualMode_SW" THEN
       RESET_TIMER("Drill_OperationTP");
       RESET_TIMER("Mix_OperationTP");
       RESET_TIMER("Drill_PostTP");
       RESET_TIMER("Mix_PostTP");
   END_IF;
END_REGION

REGION Network 8: Pusher #2
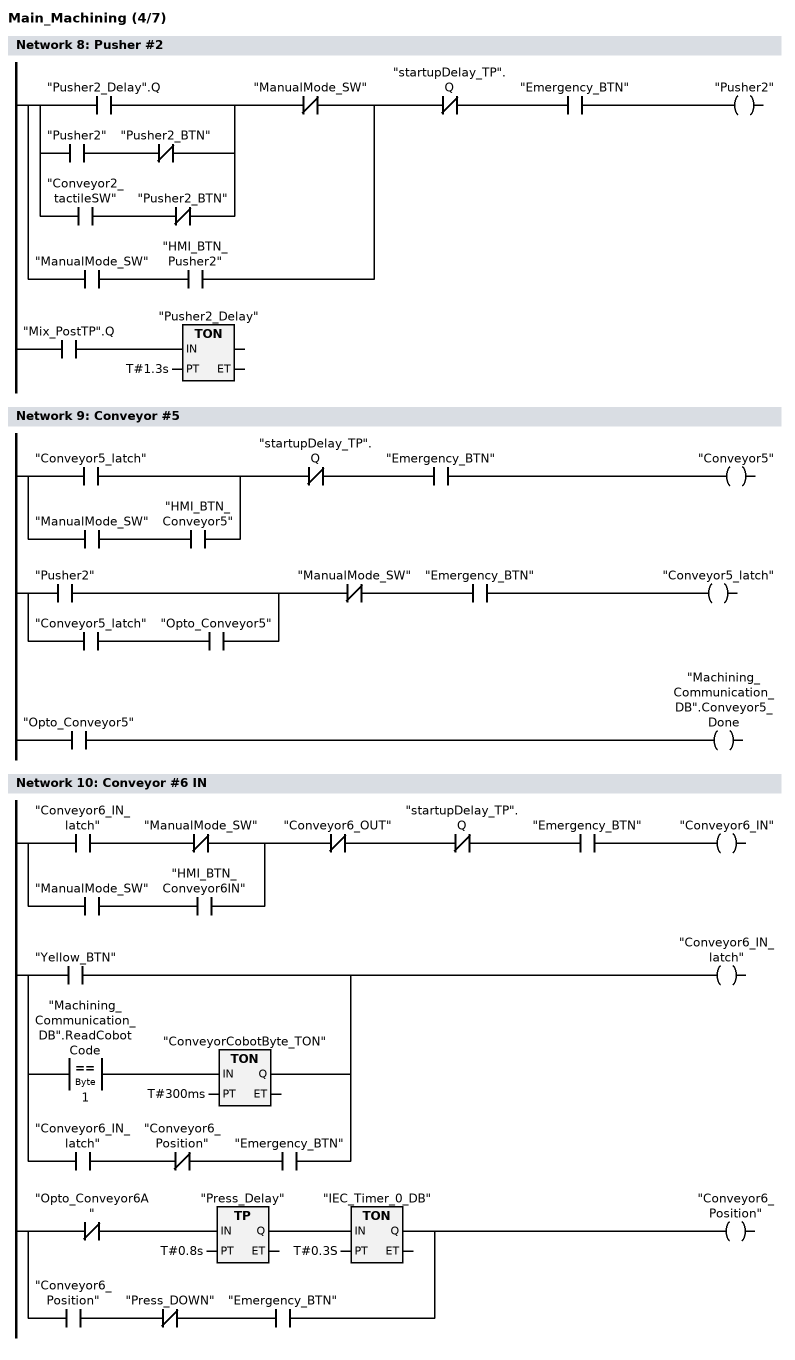
   "Pusher2" := ((("Pusher2_Delay".Q OR ("Pusher2" AND NOT "Pusher2_BTN") OR ("Conveyor2_tactileSW" AND NOT "Pusher2_BTN")) AND NOT "ManualMode_SW") OR ("ManualMode_SW" AND "HMI_BTN_Pusher2")) AND NOT "startupDelay_TP".Q AND "Emergency_BTN";
   "Pusher2_Delay".TON(IN := "Mix_PostTP".Q, PT := T#1.3s);
END_REGION

REGION Network 9: Conveyor #5
   RUNG wire#powerrail
      Contact( "Conveyor5_latch" )
      wire#w1
      I_Contact( "startupDelay_TP".Q )
      Contact( "Emergency_BTN" )
      Coil( "Conveyor5" )
   END_RUNG
   RUNG wire#powerrail
      Contact( "ManualMode_SW" )
      Contact( "HMI_BTN_Conveyor5" )
   END_RUNG wire#w1
   RUNG wire#powerrail
      Contact( "Pusher2" )
      wire#w2
      I_Contact( "ManualMode_SW" )
      Contact( "Emergency_BTN" )
      Coil( "Conveyor5_latch" )
   END_RUNG
   RUNG wire#powerrail
      Contact( "Conveyor5_latch" )
      Contact( "Opto_Conveyor5" )
   END_RUNG wire#w2
   RUNG wire#powerrail
      Contact( "Opto_Conveyor5" )
      Coil( "Machining_Communication_DB".Conveyor5_Done )
   END_RUNG
   // the same network as SCL:
   "Conveyor5" := ("Conveyor5_latch" OR ("ManualMode_SW" AND "HMI_BTN_Conveyor5")) AND NOT "startupDelay_TP".Q AND "Emergency_BTN";
   "Conveyor5_latch" := ("Pusher2" OR ("Conveyor5_latch" AND "Opto_Conveyor5")) AND NOT "ManualMode_SW" AND "Emergency_BTN";
   "Machining_Communication_DB".Conveyor5_Done := "Opto_Conveyor5";
END_REGION

REGION Network 10: Conveyor #6 IN
   "Conveyor6_IN" := (("Conveyor6_IN_latch" AND NOT "ManualMode_SW") OR ("ManualMode_SW" AND "HMI_BTN_Conveyor6IN")) AND NOT "Conveyor6_OUT" AND NOT "startupDelay_TP".Q AND "Emergency_BTN";
   "ConveyorCobotByte_TON".TON(IN := "Machining_Communication_DB".ReadCobotCode = 1, PT := T#300ms);
   "Conveyor6_IN_latch" := "Yellow_BTN" OR "ConveyorCobotByte_TON".Q OR ("Conveyor6_IN_latch" AND NOT "Conveyor6_Position" AND "Emergency_BTN");
   "Press_Delay".TP(IN := NOT "Opto_Conveyor6A", PT := T#0.8s);
   "IEC_Timer_0_DB".TON(IN := "Press_Delay".Q, PT := T#0.3S);
   "Conveyor6_Position" := "IEC_Timer_0_DB".Q OR ("Conveyor6_Position" AND NOT "Press_DOWN" AND "Emergency_BTN");
END_REGION

REGION Network 11: Press
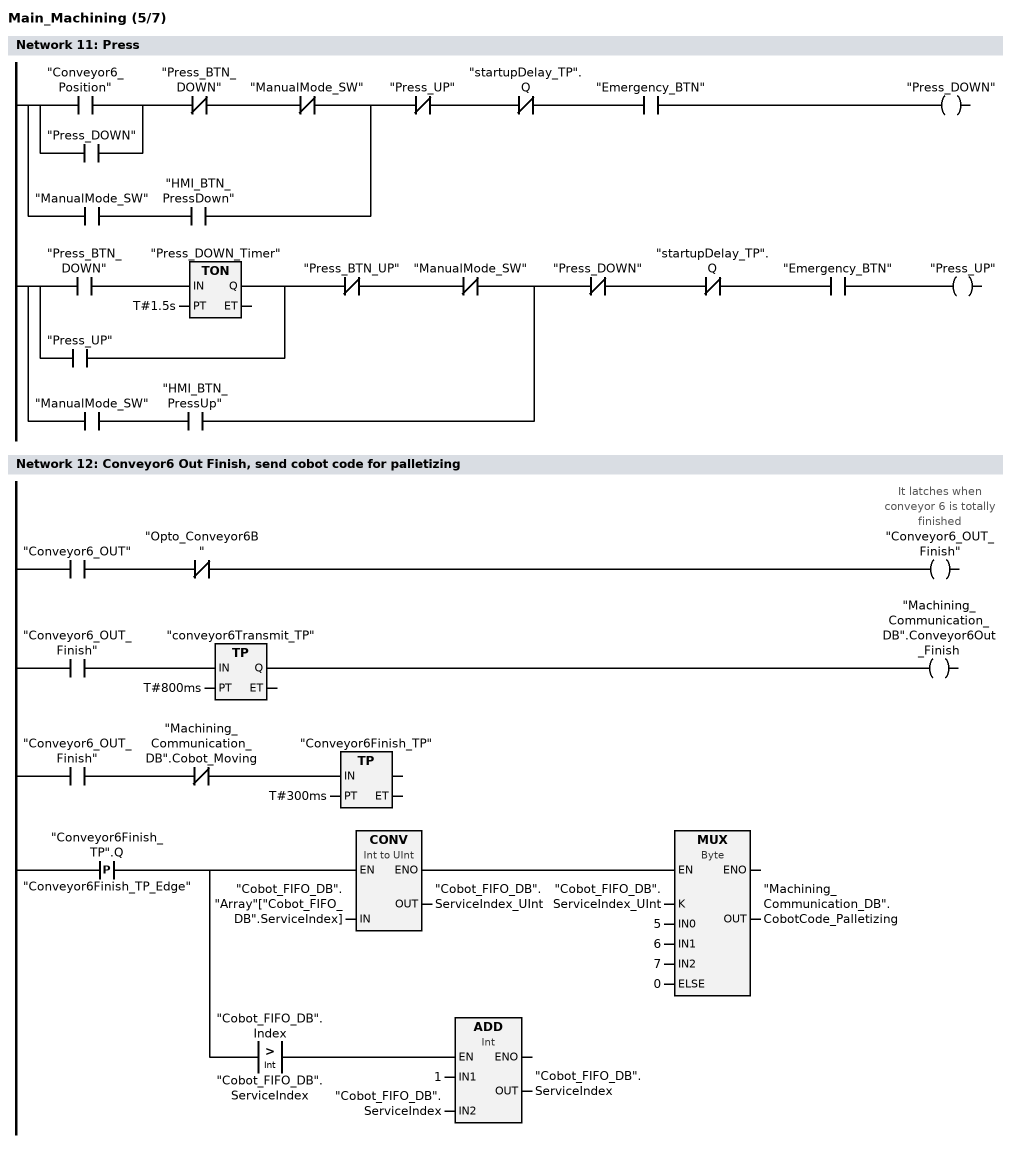
   "Press_DOWN" := ((("Conveyor6_Position" OR "Press_DOWN") AND NOT "Press_BTN_DOWN" AND NOT "ManualMode_SW") OR ("ManualMode_SW" AND "HMI_BTN_PressDown")) AND NOT "Press_UP" AND NOT "startupDelay_TP".Q AND "Emergency_BTN";
   "Press_DOWN_Timer".TON(IN := "Press_BTN_DOWN", PT := T#1.5s);
   "Press_UP" := ((("Press_DOWN_Timer".Q OR "Press_UP") AND NOT "Press_BTN_UP" AND NOT "ManualMode_SW") OR ("ManualMode_SW" AND "HMI_BTN_PressUp")) AND NOT "Press_DOWN" AND NOT "startupDelay_TP".Q AND "Emergency_BTN";
END_REGION

REGION Network 12: Conveyor6 Out Finish, send cobot code for palletizing
   // no SCL statement known for Mux: written as a call
   "Conveyor6_OUT_Finish" := "Conveyor6_OUT" AND NOT "Opto_Conveyor6B";   // It latches when conveyor 6 is totally finished
   "conveyor6Transmit_TP".TP(IN := "Conveyor6_OUT_Finish", PT := T#800ms);
   "Machining_Communication_DB".Conveyor6Out_Finish := "conveyor6Transmit_TP".Q;
   "Conveyor6Finish_TP".TP(IN := "Conveyor6_OUT_Finish" AND NOT "Machining_Communication_DB".Cobot_Moving,
                           PT := T#300ms);
   #_w1 := "Conveyor6Finish_TP".Q AND NOT "Conveyor6Finish_TP_Edge";   // rising edge of "Conveyor6Finish_TP".Q
   "Conveyor6Finish_TP_Edge" := "Conveyor6Finish_TP".Q;
   IF #_w1 THEN
       "Cobot_FIFO_DB".ServiceIndex_UInt := INT_TO_UINT("Cobot_FIFO_DB"."Array"["Cobot_FIFO_DB".ServiceIndex]);
       Mux(k := "Cobot_FIFO_DB".ServiceIndex_UInt,
           in0 := 5,
           in1 := 6,
           in2 := 7,
           "else" := 0,
           out => "Machining_Communication_DB".CobotCode_Palletizing);
   END_IF;
   IF #_w1 AND ("Cobot_FIFO_DB".Index > "Cobot_FIFO_DB".ServiceIndex) THEN
       "Cobot_FIFO_DB".ServiceIndex := 1 + "Cobot_FIFO_DB".ServiceIndex;
   END_IF;
END_REGION

REGION Network 13: Reset FIFO when logout
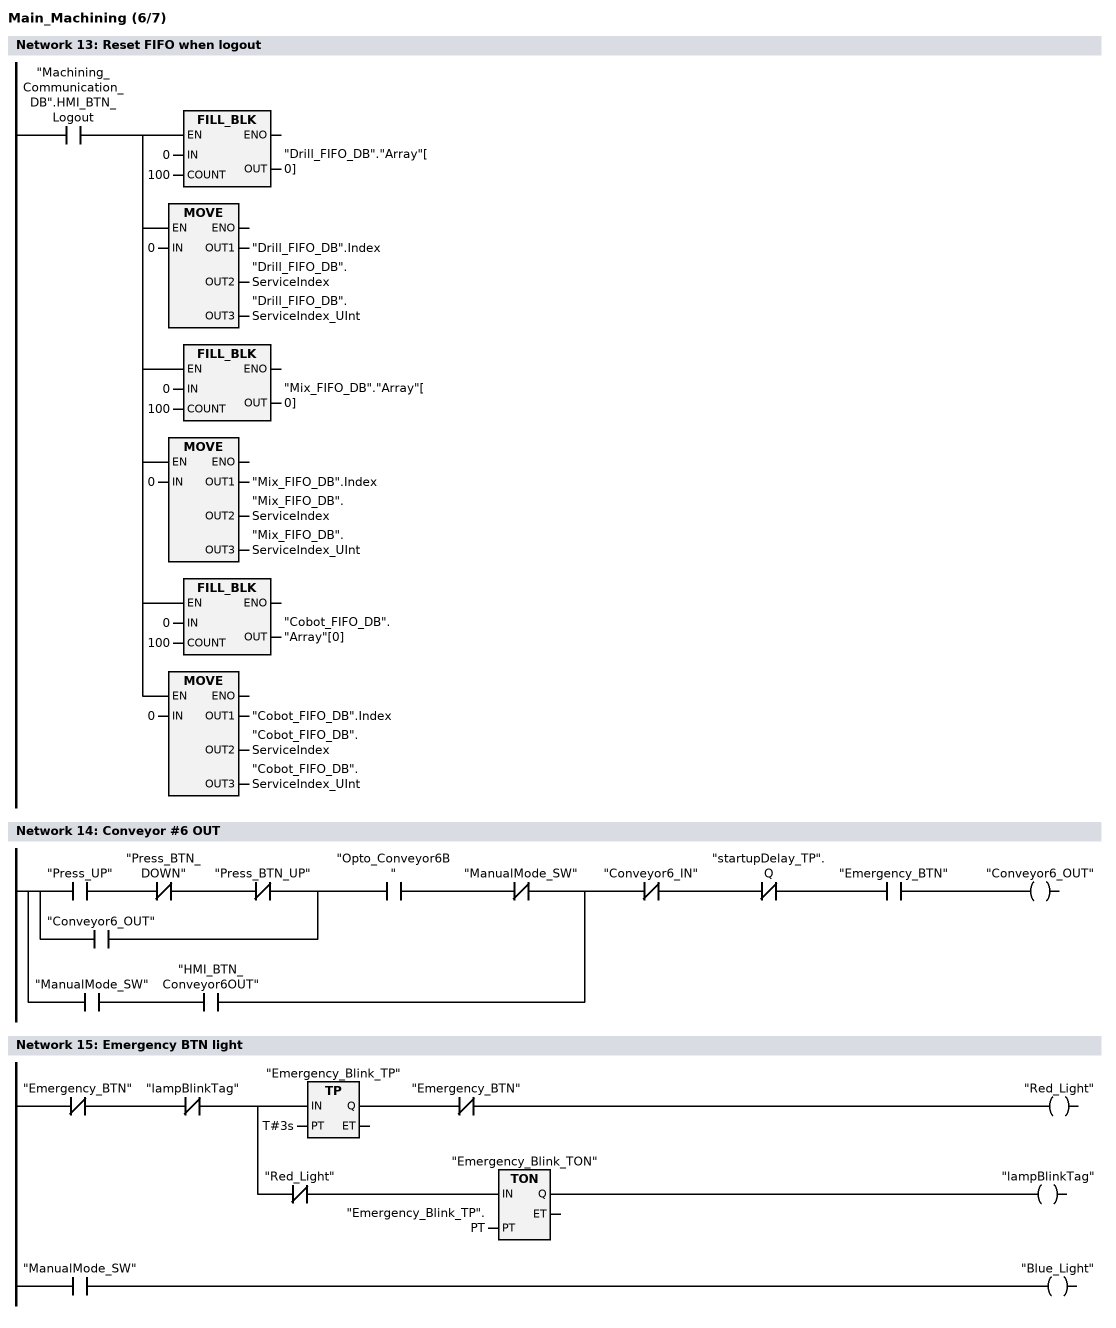
   RUNG wire#powerrail
      Contact( "Machining_Communication_DB".HMI_BTN_Logout )
      wire#w1
      FillBlockI(in := 0, count := 100, out => "Drill_FIFO_DB"."Array"[0])
   END_RUNG
   RUNG wire#w1
      Move(in := 0, out1 => "Drill_FIFO_DB".Index, out2 => "Drill_FIFO_DB".ServiceIndex, out3 => "Drill_FIFO_DB".ServiceIndex_UInt)
   END_RUNG
   RUNG wire#w1
      FillBlockI(in := 0, count := 100, out => "Mix_FIFO_DB"."Array"[0])
   END_RUNG
   RUNG wire#w1
      Move(in := 0, out1 => "Mix_FIFO_DB".Index, out2 => "Mix_FIFO_DB".ServiceIndex, out3 => "Mix_FIFO_DB".ServiceIndex_UInt)
   END_RUNG
   RUNG wire#w1
      FillBlockI(in := 0, count := 100, out => "Cobot_FIFO_DB"."Array"[0])
   END_RUNG
   RUNG wire#w1
      Move(in := 0, out1 => "Cobot_FIFO_DB".Index, out2 => "Cobot_FIFO_DB".ServiceIndex, out3 => "Cobot_FIFO_DB".ServiceIndex_UInt)
   END_RUNG
   // the same network as SCL:
   #_w1 := "Machining_Communication_DB".HMI_BTN_Logout;
   IF #_w1 THEN
       FILL_BLK(IN := 0, COUNT := 100, OUT => "Drill_FIFO_DB"."Array"[0]);
       "Drill_FIFO_DB".Index := 0;
       "Drill_FIFO_DB".ServiceIndex := 0;
       "Drill_FIFO_DB".ServiceIndex_UInt := 0;
       FILL_BLK(IN := 0, COUNT := 100, OUT => "Mix_FIFO_DB"."Array"[0]);
       "Mix_FIFO_DB".Index := 0;
       "Mix_FIFO_DB".ServiceIndex := 0;
       "Mix_FIFO_DB".ServiceIndex_UInt := 0;
       FILL_BLK(IN := 0, COUNT := 100, OUT => "Cobot_FIFO_DB"."Array"[0]);
       "Cobot_FIFO_DB".Index := 0;
       "Cobot_FIFO_DB".ServiceIndex := 0;
       "Cobot_FIFO_DB".ServiceIndex_UInt := 0;
   END_IF;
END_REGION

REGION Network 14: Conveyor #6 OUT
   RUNG wire#powerrail
      Contact( "Press_UP" )
      I_Contact( "Press_BTN_DOWN" )
      I_Contact( "Press_BTN_UP" )
      wire#w1
      Contact( "Opto_Conveyor6B" )
      I_Contact( "ManualMode_SW" )
      wire#w2
      I_Contact( "Conveyor6_IN" )
      I_Contact( "startupDelay_TP".Q )
      Contact( "Emergency_BTN" )
      Coil( "Conveyor6_OUT" )
   END_RUNG
   RUNG wire#powerrail
      Contact( "Conveyor6_OUT" )
   END_RUNG wire#w1
   RUNG wire#powerrail
      Contact( "ManualMode_SW" )
      Contact( "HMI_BTN_Conveyor6OUT" )
   END_RUNG wire#w2
   // the same network as SCL:
   "Conveyor6_OUT" := (((("Press_UP" AND NOT "Press_BTN_DOWN" AND NOT "Press_BTN_UP") OR "Conveyor6_OUT") AND "Opto_Conveyor6B" AND NOT "ManualMode_SW") OR ("ManualMode_SW" AND "HMI_BTN_Conveyor6OUT")) AND NOT "Conveyor6_IN" AND NOT "startupDelay_TP".Q AND "Emergency_BTN";
END_REGION

REGION Network 15: Emergency BTN light
   #_w1 := NOT "Emergency_BTN" AND NOT "lampBlinkTag";
   "Emergency_Blink_TP".TP(IN := #_w1, PT := T#3s);
   "Red_Light" := "Emergency_Blink_TP".Q AND NOT "Emergency_BTN";
   "Emergency_Blink_TON".TON(IN := #_w1 AND NOT "Red_Light", PT := "Emergency_Blink_TP".PT);
   "lampBlinkTag" := "Emergency_Blink_TON".Q;
   "Blue_Light" := "ManualMode_SW";
END_REGION

REGION Network 16: Read cell potentiometer
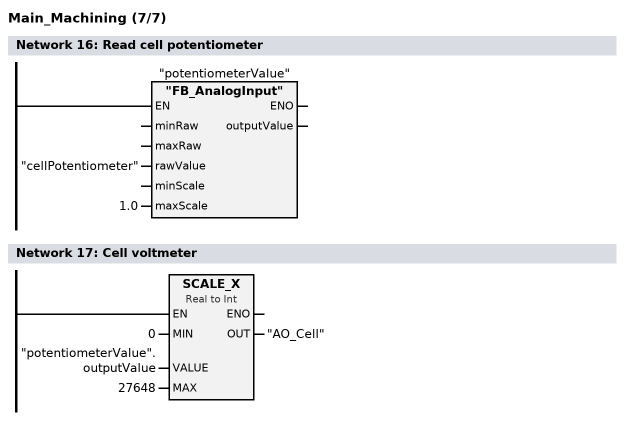
   RUNG wire#powerrail
      "potentiometerValue"(minRaw :=, maxRaw :=, rawValue := "cellPotentiometer", minScale :=, maxScale := 1.0, outputValue =>)
   END_RUNG
   // the same network as SCL:
   "potentiometerValue"(rawValue := "cellPotentiometer", maxScale := 1.0);   // "FB_AnalogInput"
END_REGION

REGION Network 17: Cell voltmeter
   RUNG wire#powerrail
      { S7_Templates := "[SrcType := Real, DestType := Int]" } Scale(min := 0, value := "potentiometerValue".outputValue, max := 27648, out => "AO_Cell")
   END_RUNG
   // the same network as SCL:
   "AO_Cell" := SCALE_X(MIN := 0, VALUE := "potentiometerValue".outputValue, MAX := 27648);
END_REGION
END_ORGANIZATION_BLOCK

ORGANIZATION_BLOCK "HMI_OB"   // OB123, LAD, ProgramCycle
{ S7_Optimized_Access := 'TRUE' }
VERSION : 0.1
   VAR_INPUT
      Initial_Call : Bool;
      Remanence : Bool;
   END_VAR
BEGIN

REGION Network 1: Set access screen at program startup
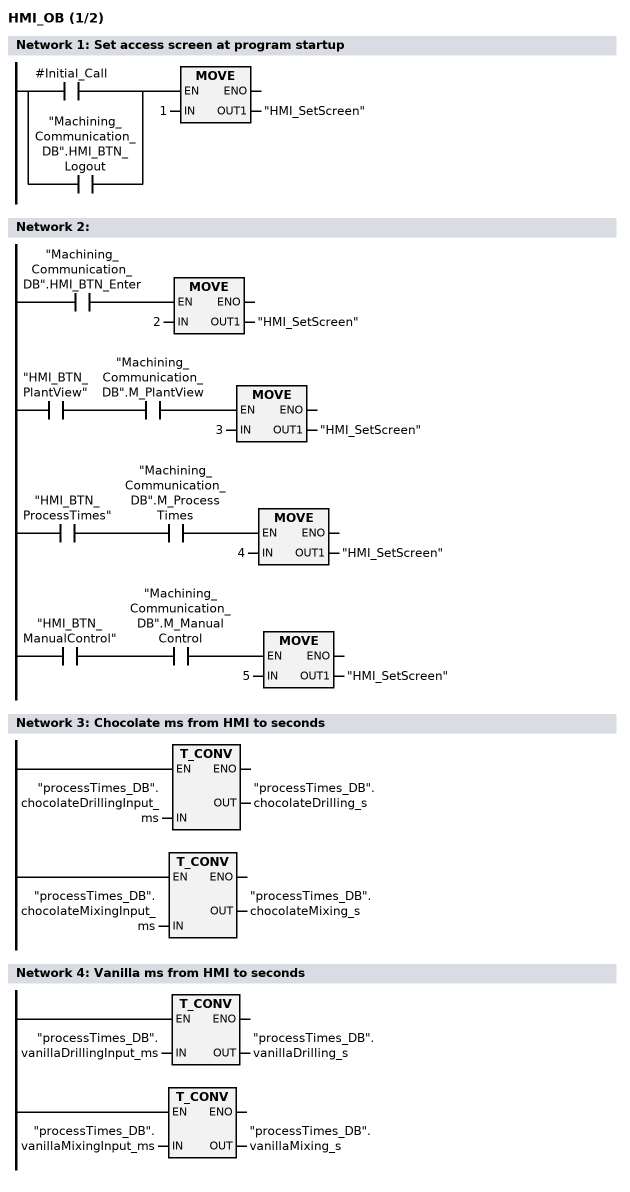
   RUNG wire#powerrail
      Contact( #Initial_Call )
      wire#w1
      Move(in := 1, out1 => "HMI_SetScreen")
   END_RUNG
   RUNG wire#powerrail
      Contact( "Machining_Communication_DB".HMI_BTN_Logout )
   END_RUNG wire#w1
   // the same network as SCL:
   IF #Initial_Call OR "Machining_Communication_DB".HMI_BTN_Logout THEN "HMI_SetScreen" := 1; END_IF;
END_REGION

REGION Network 2
   RUNG wire#powerrail
      Contact( "Machining_Communication_DB".HMI_BTN_Enter )
      Move(in := 2, out1 => "HMI_SetScreen")
   END_RUNG
   RUNG wire#powerrail
      Contact( "HMI_BTN_PlantView" )
      Contact( "Machining_Communication_DB".M_PlantView )
      Move(in := 3, out1 => "HMI_SetScreen")
   END_RUNG
   RUNG wire#powerrail
      Contact( "HMI_BTN_ProcessTimes" )
      Contact( "Machining_Communication_DB".M_ProcessTimes )
      Move(in := 4, out1 => "HMI_SetScreen")
   END_RUNG
   RUNG wire#powerrail
      Contact( "HMI_BTN_ManualControl" )
      Contact( "Machining_Communication_DB".M_ManualControl )
      Move(in := 5, out1 => "HMI_SetScreen")
   END_RUNG
   // the same network as SCL:
   IF "Machining_Communication_DB".HMI_BTN_Enter THEN "HMI_SetScreen" := 2; END_IF;
   IF "HMI_BTN_PlantView" AND "Machining_Communication_DB".M_PlantView THEN "HMI_SetScreen" := 3; END_IF;
   IF "HMI_BTN_ProcessTimes" AND "Machining_Communication_DB".M_ProcessTimes THEN
       "HMI_SetScreen" := 4;
   END_IF;
   IF "HMI_BTN_ManualControl" AND "Machining_Communication_DB".M_ManualControl THEN
       "HMI_SetScreen" := 5;
   END_IF;
END_REGION

REGION Network 3: Chocolate ms from HMI to seconds
   "processTimes_DB".chocolateDrilling_s := T_CONV(IN := "processTimes_DB".chocolateDrillingInput_ms);
   "processTimes_DB".chocolateMixing_s := T_CONV(IN := "processTimes_DB".chocolateMixingInput_ms);
END_REGION

REGION Network 4: Vanilla ms from HMI to seconds
   "processTimes_DB".vanillaDrilling_s := T_CONV(IN := "processTimes_DB".vanillaDrillingInput_ms);
   "processTimes_DB".vanillaMixing_s := T_CONV(IN := "processTimes_DB".vanillaMixingInput_ms);
END_REGION

REGION Network 5: Strawberry ms from HMI to seconds
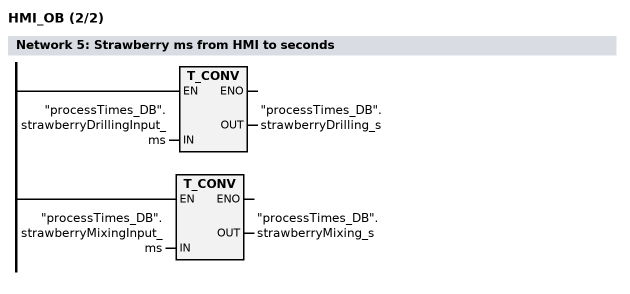
   "processTimes_DB".strawberryDrilling_s := T_CONV(IN := "processTimes_DB".strawberryDrillingInput_ms);
   "processTimes_DB".strawberryMixing_s := T_CONV(IN := "processTimes_DB".strawberryMixingInput_ms);
END_REGION
END_ORGANIZATION_BLOCK

ORGANIZATION_BLOCK "Cognex_OB"   // OB124, LAD, ProgramCycle
{ S7_Optimized_Access := 'TRUE' }
VERSION : 0.1
   VAR_INPUT
      Initial_Call : Bool;
      Remanence : Bool;
   END_VAR
BEGIN

REGION Network 1: Set the cognex ID and code to -1 on startup
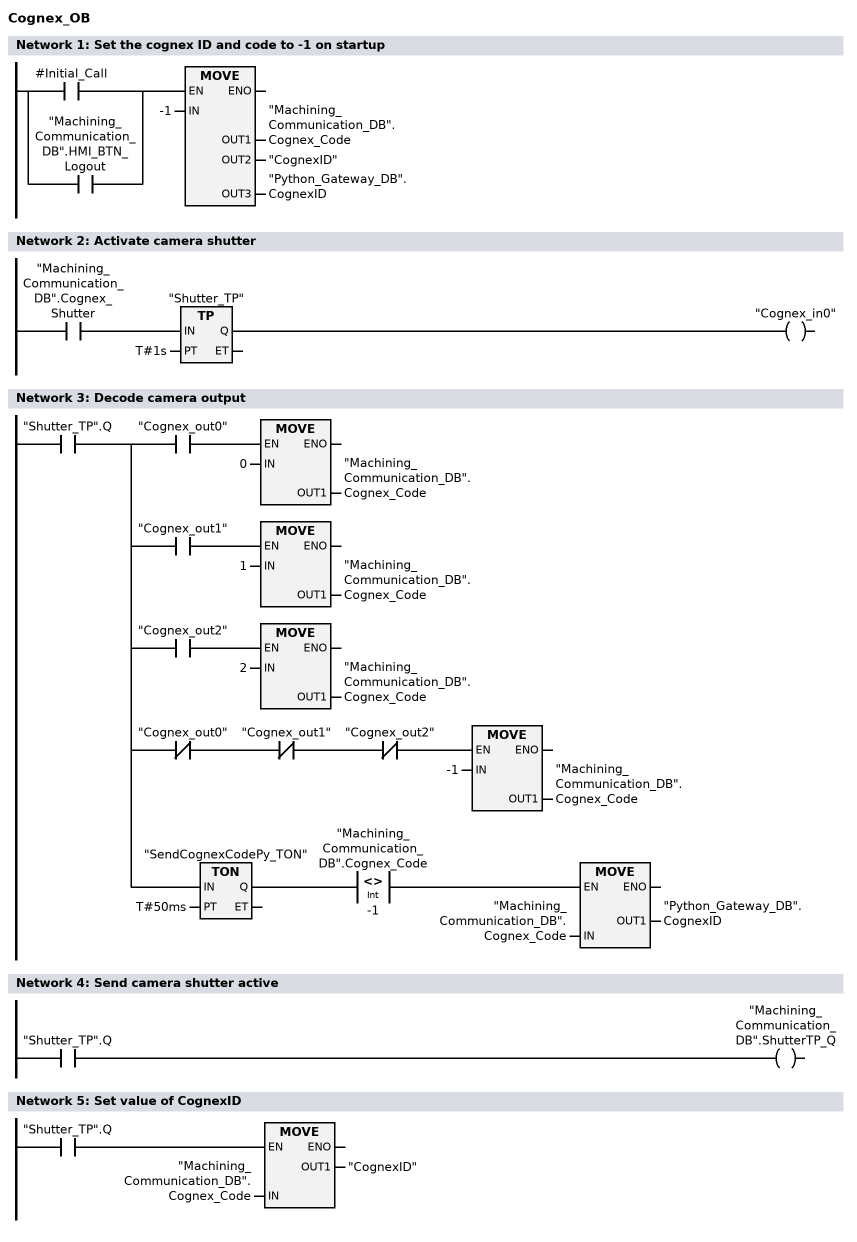
   RUNG wire#powerrail
      Contact( #Initial_Call )
      wire#w1
      Move(in := -1, out1 => "Machining_Communication_DB".Cognex_Code, out2 => "CognexID", out3 => "Python_Gateway_DB".CognexID)
   END_RUNG
   RUNG wire#powerrail
      Contact( "Machining_Communication_DB".HMI_BTN_Logout )
   END_RUNG wire#w1
   // the same network as SCL:
   IF #Initial_Call OR "Machining_Communication_DB".HMI_BTN_Logout THEN
       "Machining_Communication_DB".Cognex_Code := -1;
       "CognexID" := -1;
       "Python_Gateway_DB".CognexID := -1;
   END_IF;
END_REGION

REGION Network 2: Activate camera shutter
   "Shutter_TP".TP(IN := "Machining_Communication_DB".Cognex_Shutter, PT := T#1s);
   "Cognex_in0" := "Shutter_TP".Q;
END_REGION

REGION Network 3: Decode camera output
   IF "Shutter_TP".Q AND "Cognex_out0" THEN "Machining_Communication_DB".Cognex_Code := 0; END_IF;
   IF "Shutter_TP".Q AND "Cognex_out1" THEN "Machining_Communication_DB".Cognex_Code := 1; END_IF;
   IF "Shutter_TP".Q AND "Cognex_out2" THEN "Machining_Communication_DB".Cognex_Code := 2; END_IF;
   IF "Shutter_TP".Q AND NOT "Cognex_out0" AND NOT "Cognex_out1" AND NOT "Cognex_out2" THEN
       "Machining_Communication_DB".Cognex_Code := -1;
   END_IF;
   "SendCognexCodePy_TON".TON(IN := "Shutter_TP".Q, PT := T#50ms);
   IF "SendCognexCodePy_TON".Q AND ("Machining_Communication_DB".Cognex_Code <> (-1)) THEN
       "Python_Gateway_DB".CognexID := "Machining_Communication_DB".Cognex_Code;
   END_IF;
END_REGION

REGION Network 4: Send camera shutter active
   RUNG wire#powerrail
      Contact( "Shutter_TP".Q )
      Coil( "Machining_Communication_DB".ShutterTP_Q )
   END_RUNG
   // the same network as SCL:
   "Machining_Communication_DB".ShutterTP_Q := "Shutter_TP".Q;
END_REGION

REGION Network 5: Set value of CognexID
   RUNG wire#powerrail
      Contact( "Shutter_TP".Q )
      Move(in := "Machining_Communication_DB".Cognex_Code, out1 => "CognexID")
   END_RUNG
   // the same network as SCL:
   IF "Shutter_TP".Q THEN "CognexID" := "Machining_Communication_DB".Cognex_Code; END_IF;
END_REGION
END_ORGANIZATION_BLOCK

ORGANIZATION_BLOCK "Monitoring_OB"   // OB125, LAD, ProgramCycle
{ S7_Optimized_Access := 'TRUE' }
VERSION : 0.1
   VAR_INPUT
      Initial_Call : Bool;
      Remanence : Bool;
   END_VAR
BEGIN

REGION Network 1: Measure power consumption
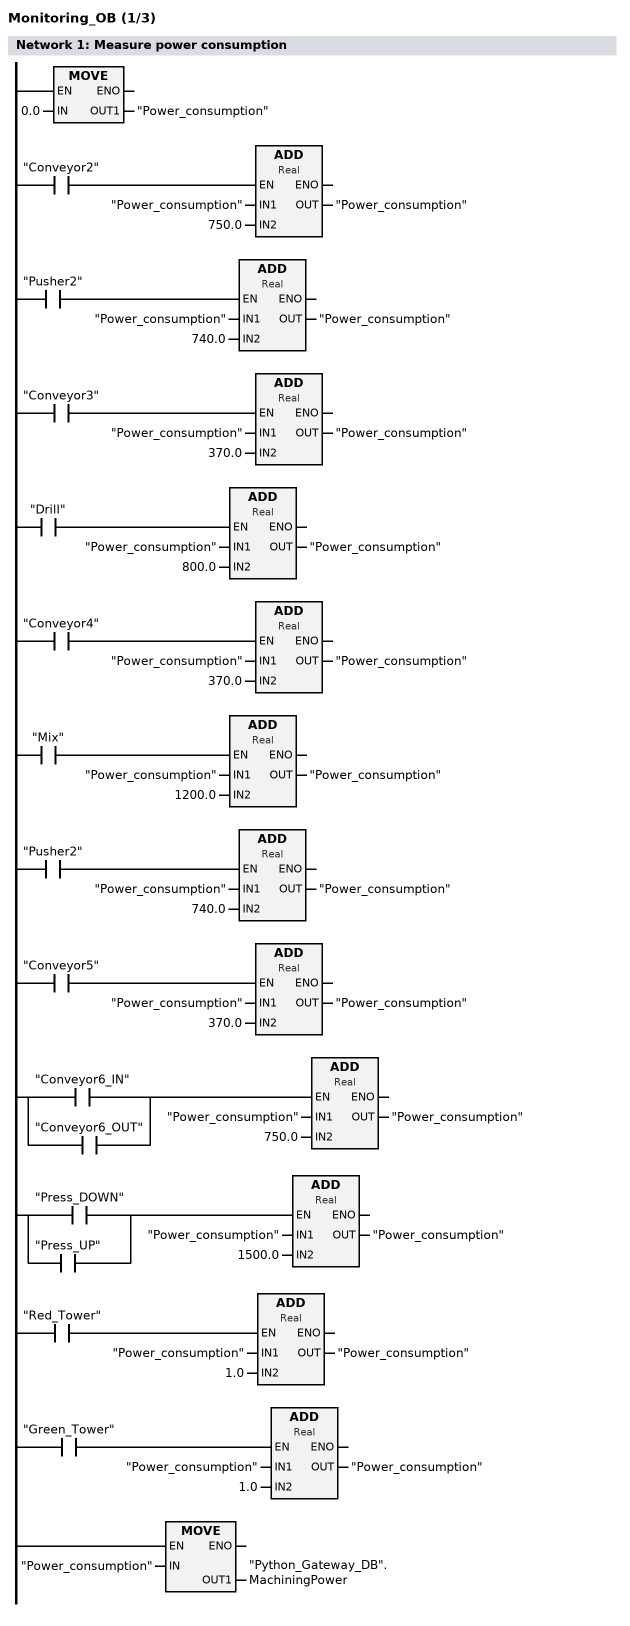
   RUNG wire#powerrail
      Move(in := 0.0, out1 => "Power_consumption")
   END_RUNG
   RUNG wire#powerrail
      Contact( "Conveyor2" )
      { S7_Templates := "SrcType := Real" } Add(in1 := "Power_consumption", in2 := 750.0, out => "Power_consumption")
   END_RUNG
   RUNG wire#powerrail
      Contact( "Pusher2" )
      { S7_Templates := "SrcType := Real" } Add(in1 := "Power_consumption", in2 := 740.0, out => "Power_consumption")
   END_RUNG
   RUNG wire#powerrail
      Contact( "Conveyor3" )
      { S7_Templates := "SrcType := Real" } Add(in1 := "Power_consumption", in2 := 370.0, out => "Power_consumption")
   END_RUNG
   RUNG wire#powerrail
      Contact( "Drill" )
      { S7_Templates := "SrcType := Real" } Add(in1 := "Power_consumption", in2 := 800.0, out => "Power_consumption")
   END_RUNG
   RUNG wire#powerrail
      Contact( "Conveyor4" )
      { S7_Templates := "SrcType := Real" } Add(in1 := "Power_consumption", in2 := 370.0, out => "Power_consumption")
   END_RUNG
   RUNG wire#powerrail
      Contact( "Mix" )
      { S7_Templates := "SrcType := Real" } Add(in1 := "Power_consumption", in2 := 1200.0, out => "Power_consumption")
   END_RUNG
   RUNG wire#powerrail
      Contact( "Pusher2" )
      { S7_Templates := "SrcType := Real" } Add(in1 := "Power_consumption", in2 := 740.0, out => "Power_consumption")
   END_RUNG
   RUNG wire#powerrail
      Contact( "Conveyor5" )
      { S7_Templates := "SrcType := Real" } Add(in1 := "Power_consumption", in2 := 370.0, out => "Power_consumption")
   END_RUNG
   RUNG wire#powerrail
      Contact( "Conveyor6_IN" )
      wire#w1
      { S7_Templates := "SrcType := Real" } Add(in1 := "Power_consumption", in2 := 750.0, out => "Power_consumption")
   END_RUNG
   RUNG wire#powerrail
      Contact( "Conveyor6_OUT" )
   END_RUNG wire#w1
   RUNG wire#powerrail
      Contact( "Press_DOWN" )
      wire#w2
      { S7_Templates := "SrcType := Real" } Add(in1 := "Power_consumption", in2 := 1500.0, out => "Power_consumption")
   END_RUNG
   RUNG wire#powerrail
      Contact( "Press_UP" )
   END_RUNG wire#w2
   RUNG wire#powerrail
      Contact( "Red_Tower" )
      { S7_Templates := "SrcType := Real" } Add(in1 := "Power_consumption", in2 := 1.0, out => "Power_consumption")
   END_RUNG
   RUNG wire#powerrail
      Contact( "Green_Tower" )
      { S7_Templates := "SrcType := Real" } Add(in1 := "Power_consumption", in2 := 1.0, out => "Power_consumption")
   END_RUNG
   RUNG wire#powerrail
      Move(in := "Power_consumption", out1 => "Python_Gateway_DB".MachiningPower)
   END_RUNG
   // the same network as SCL:
   "Power_consumption" := 0.0;
   IF "Conveyor2" THEN "Power_consumption" := "Power_consumption" + 750.0; END_IF;
   IF "Pusher2" THEN "Power_consumption" := "Power_consumption" + 740.0; END_IF;
   IF "Conveyor3" THEN "Power_consumption" := "Power_consumption" + 370.0; END_IF;
   IF "Drill" THEN "Power_consumption" := "Power_consumption" + 800.0; END_IF;
   IF "Conveyor4" THEN "Power_consumption" := "Power_consumption" + 370.0; END_IF;
   IF "Mix" THEN "Power_consumption" := "Power_consumption" + 1200.0; END_IF;
   IF "Pusher2" THEN "Power_consumption" := "Power_consumption" + 740.0; END_IF;
   IF "Conveyor5" THEN "Power_consumption" := "Power_consumption" + 370.0; END_IF;
   IF "Conveyor6_IN" OR "Conveyor6_OUT" THEN "Power_consumption" := "Power_consumption" + 750.0; END_IF;
   IF "Press_DOWN" OR "Press_UP" THEN "Power_consumption" := "Power_consumption" + 1500.0; END_IF;
   IF "Red_Tower" THEN "Power_consumption" := "Power_consumption" + 1.0; END_IF;
   IF "Green_Tower" THEN "Power_consumption" := "Power_consumption" + 1.0; END_IF;
   "Python_Gateway_DB".MachiningPower := "Power_consumption";
END_REGION

REGION Network 2: Send emergency BTNs to Python Gateway
   // Contact is negated, when BTN is pressed, the DB bit turns true
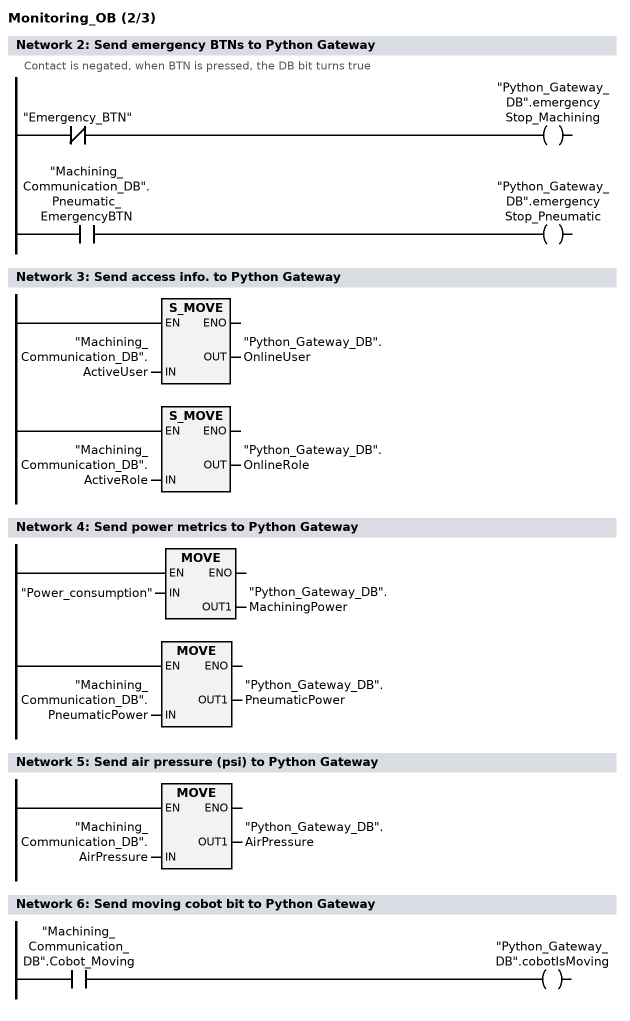
   RUNG wire#powerrail
      I_Contact( "Emergency_BTN" )
      Coil( "Python_Gateway_DB".emergencyStop_Machining )
   END_RUNG
   RUNG wire#powerrail
      Contact( "Machining_Communication_DB".Pneumatic_EmergencyBTN )
      Coil( "Python_Gateway_DB".emergencyStop_Pneumatic )
   END_RUNG
   // the same network as SCL:
   "Python_Gateway_DB".emergencyStop_Machining := NOT "Emergency_BTN";
   "Python_Gateway_DB".emergencyStop_Pneumatic := "Machining_Communication_DB".Pneumatic_EmergencyBTN;
END_REGION

REGION Network 3: Send access info. to Python Gateway
   RUNG wire#powerrail
      S_Move(in := "Machining_Communication_DB".ActiveUser, out => "Python_Gateway_DB".OnlineUser)
   END_RUNG
   RUNG wire#powerrail
      S_Move(in := "Machining_Communication_DB".ActiveRole, out => "Python_Gateway_DB".OnlineRole)
   END_RUNG
   // the same network as SCL:
   "Python_Gateway_DB".OnlineUser := "Machining_Communication_DB".ActiveUser;
   "Python_Gateway_DB".OnlineRole := "Machining_Communication_DB".ActiveRole;
END_REGION

REGION Network 4: Send power metrics to Python Gateway
   RUNG wire#powerrail
      Move(in := "Power_consumption", out1 => "Python_Gateway_DB".MachiningPower)
   END_RUNG
   RUNG wire#powerrail
      Move(in := "Machining_Communication_DB".PneumaticPower, out1 => "Python_Gateway_DB".PneumaticPower)
   END_RUNG
   // the same network as SCL:
   "Python_Gateway_DB".MachiningPower := "Power_consumption";
   "Python_Gateway_DB".PneumaticPower := "Machining_Communication_DB".PneumaticPower;
END_REGION

REGION Network 5: Send air pressure (psi) to Python Gateway
   RUNG wire#powerrail
      Move(in := "Machining_Communication_DB".AirPressure, out1 => "Python_Gateway_DB".AirPressure)
   END_RUNG
   // the same network as SCL:
   "Python_Gateway_DB".AirPressure := "Machining_Communication_DB".AirPressure;
END_REGION

REGION Network 6: Send moving cobot bit to Python Gateway
   RUNG wire#powerrail
      Contact( "Machining_Communication_DB".Cobot_Moving )
      Coil( "Python_Gateway_DB".cobotIsMoving )
   END_RUNG
   // the same network as SCL:
   "Python_Gateway_DB".cobotIsMoving := "Machining_Communication_DB".Cobot_Moving;
END_REGION

REGION Network 7: Send finished units to Python Gateway
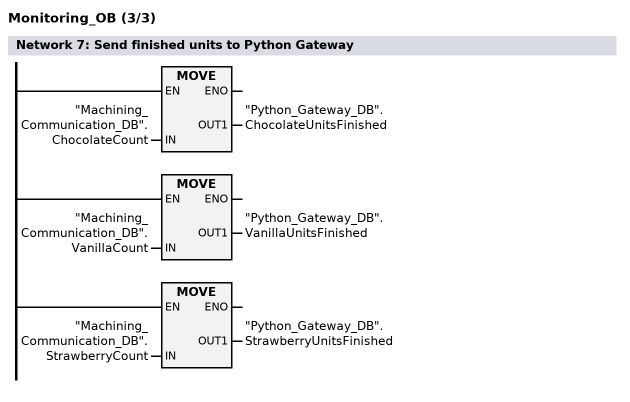
   RUNG wire#powerrail
      Move(in := "Machining_Communication_DB".ChocolateCount, out1 => "Python_Gateway_DB".ChocolateUnitsFinished)
   END_RUNG
   RUNG wire#powerrail
      Move(in := "Machining_Communication_DB".VanillaCount, out1 => "Python_Gateway_DB".VanillaUnitsFinished)
   END_RUNG
   RUNG wire#powerrail
      Move(in := "Machining_Communication_DB".StrawberryCount, out1 => "Python_Gateway_DB".StrawberryUnitsFinished)
   END_RUNG
   // the same network as SCL:
   "Python_Gateway_DB".ChocolateUnitsFinished := "Machining_Communication_DB".ChocolateCount;
   "Python_Gateway_DB".VanillaUnitsFinished := "Machining_Communication_DB".VanillaCount;
   "Python_Gateway_DB".StrawberryUnitsFinished := "Machining_Communication_DB".StrawberryCount;
END_REGION
END_ORGANIZATION_BLOCK

// ===== PLC "PLC_Pneumatic"  CPU 1214C AC/DC/Rly =====

VAR_GLOBAL   // PLC tag table "Default tag table"
   "normPressure" AT %MD30 : Real;
   "pressureValue" AT %MD34 : Real;
   "cakeFlavor" AT %MW38 : UInt;
   "PunchingTime" AT %MD40 : Time;
   "CognexId_UInt" AT %MW10 : UInt;
   "initialPhotoPending" AT %M12.0 : Bool;
   "secondsSincePhoto" AT %MD14 : DInt;
   "ReceiveCognexID_Edge" AT %M18.0 : Bool;
   "PneumaticStationBusy" AT %M18.1 : Bool;
   "Power_consumption" AT %MD44 : Real;
   "CognexID" AT %MW20 : Int;
END_VAR

VAR_GLOBAL   // PLC tag table "P_Cell_Tags"
   "Red_BTN" AT %I9.6 : Bool;
   "Green_BTN" AT %I9.4 : Bool;
   "Yellow_BTN" AT %I9.5 : Bool;
   "Emergency_BTN" AT %I9.7 : Bool;
   "Opto_Start" AT %I8.0 : Bool;
   "Vertical_Punch_BTN" AT %I8.1 : Bool;
   "Turntable_BTN" AT %I8.3 : Bool;
   "In_Conveyor_BTN" AT %I8.4 : Bool;
   "Opto_Conveyor_Exit1" AT %I8.5 : Bool;
   "pressureSensor" AT %IW118 : Int;
   "Red_Light" AT %Q9.6 : Bool;
   "Green_Light" AT %Q9.5 : Bool;
   "Blue_Light" AT %Q9.7 : Bool;
   "Turntable" AT %Q9.0 : Bool;
   "Conveyor1" AT %Q9.1 : Bool;
   "Ext_Piston_Start" AT %Q8.4 : Bool;
   "Cntrcn_Piston_Start" AT %Q8.3 : Bool;
   "Vertical_Piston" AT %Q8.5 : Bool;
   "Ext_Piston_Conveyor" AT %Q8.7 : Bool;
   "Cntrcn_Piston_Conveyor" AT %Q8.6 : Bool;
END_VAR

VAR_GLOBAL   // PLC tag table "Clock_Tags"
   "Clock_Byte" AT %MB0 : Byte;
   "Clock_10Hz" AT %M0.0 : Bool;
   "Clock_5Hz" AT %M0.1 : Bool;
   "Clock_2.5Hz" AT %M0.2 : Bool;
   "Clock_2Hz" AT %M0.3 : Bool;
   "Clock_1.25Hz" AT %M0.4 : Bool;
   "Clock_1Hz" AT %M0.5 : Bool;
   "Clock_0.625Hz" AT %M0.6 : Bool;
   "Clock_0.5Hz" AT %M0.7 : Bool;
END_VAR

VAR_GLOBAL   // PLC tag table "P_HMI_Tags"
   "HMI_BTN_Scan" AT %M51.2 : Bool;
   "HMI_BTN_ManualMode" AT %M51.3 : Bool;
   "HMI_BTN_Cntrcn_Piston_Conveyor" AT %M50.3 : Bool;
   "HMI_BTN_Vertical_Piston" AT %M50.4 : Bool;
   "HMI_BTN_Cntrcn_Piston_Start" AT %M50.5 : Bool;
   "HMI_BTN_Ext_Piston_Start" AT %M50.6 : Bool;
   "HMI_BTN_Ext_Piston_Conveyor" AT %M50.7 : Bool;
   "HMI_BTN_Conveyor1" AT %M51.0 : Bool;
   "HMI_BTN_Turntable" AT %M51.1 : Bool;
   "Green_BTN_HMI" AT %M50.0 : Bool;
   "Yellow_BTN_HMI" AT %M50.1 : Bool;
   "Red_BTN_HMI" AT %M50.2 : Bool;
   "HMI_ShowBusyMessage" AT %M51.4 : Bool;
   "HMI_CurrentScreen" AT %MW52 : UInt;
   "HMI_SetScreen" AT %MW54 : Int;
   "HMI_BTN_Enter" AT %M51.5 : Bool;
   "HMI_BTN_PlantView" AT %M51.6 : Bool;
   "HMI_BTN_ProcessTimes" AT %M51.7 : Bool;
   "HMI_BTN_ManualModeScr" AT %M56.0 : Bool;
   "HMI_BTN_CameraControl" AT %M56.1 : Bool;
   "HMI_BTN_Logout" AT %M56.2 : Bool;
   "HMI_BTN_CycleTime" AT %M56.3 : Bool;
   "HMI_BTN_EnableCycleTime" AT %M56.4 : Bool;
END_VAR

VAR_GLOBAL   // PLC tag table "Cobot_Tags"
   "Cobot_DI_1" AT %Q8.1 : Bool;
   "Cobot_DI_2" AT %Q8.2 : Bool;
   "Cobot_DI_3" AT %Q9.4 : Bool;
   "Stop_Moving_Cobot" AT %Q8.0 : Bool;
   "Cobot_DO_1" AT %I0.1 : Bool;
   "Cobot_DO_2" AT %I0.2 : Bool;
   "Cobot_DO_3" AT %I0.3 : Bool;
   "Cobot_Moving" AT %I0.0 : Bool;
   "ReadCobot_Byte" AT %MB8 : Byte;
   "Cobot_Byte" AT %MB9 : Byte;
   "PalletizingDone" AT %M7.0 : Bool;
   "PalletizingBusy" AT %M7.1 : Bool;
END_VAR

VAR_GLOBAL   // PLC tag table "RFID_Tags"
   "RFID_K1" AT %I9.0 : Bool;
   "RFID_K2" AT %I9.1 : Bool;
   "RFID_K3" AT %I9.2 : Bool;
   "RFID_K4" AT %I9.3 : Bool;
   "RFID_Byte" AT %MB48 : Byte;
END_VAR

DATA_BLOCK "CurrentUser_DB"   // DB11
{ S7_Optimized_Access := 'FALSE' }
VERSION : 0.1
   VAR
      UserID : USInt;
      "Name" : String[40];
      Role : String[25];
      ValidUser : Bool;
      P_PlantView : Bool;
      P_ManualControl : Bool;
      P_Camera : Bool;
      P_Cobot : Bool;
      P_ProcessTimes : Bool;
      P_CycleTime : Bool;
      M_PlantView : Bool;
      M_ManualControl : Bool;
      M_ProcessTimes : Bool;
   END_VAR
BEGIN
END_DATA_BLOCK

DATA_BLOCK "CycleTime_DB"   // DB13
{ S7_Optimized_Access := 'TRUE' }
VERSION : 0.1
   VAR
      EnabledMeasuring : Bool;
      ActiveMeasuring : Bool;
      CurrentPieceCognexID : Int;
      TargetTimeInput_ms : UInt;
      TargetTime_s : Time;
      ElapsedTime_ms : UInt;
      ElapsedTime_s : Time;
   END_VAR
BEGIN
END_DATA_BLOCK

DATA_BLOCK "Pneumatic_Times_DB"   // DB20
{ S7_Optimized_Access := 'TRUE' }
VERSION : 0.1
   VAR
      chocolatePunchingInput_ms : UInt := 2000;
      vanillaPunchingInput_ms : UInt := 4000;
      strawberryPunchingInput_ms : UInt := 6000;
      chocolatePunching_s : Time;
      vanillaPunching_s : Time;
      strawberryPunching_s : Time;
   END_VAR
BEGIN
END_DATA_BLOCK

DATA_BLOCK "Pneumatic_Communication_DB"   // DB100
{ S7_Optimized_Access := 'FALSE' }
VERSION : 0.1
   VAR
      Cognex_Code : Int;   // Machining to Pneu
      Conveyor5_Done : Bool;   // Machining to Pneu
      Conveyor2_SensorA : Bool;   // Machining to Pneu
      ShutterTP_Q : Bool;   // Machining to Pneu
      Conveyor6Out_Finish : Bool;   // Machining to Pneu
      CobotCode_Palletizing : Byte;   // Machining to Pneu
      ReadCobotCode : Byte;   // Pneu to Machining
      Cognex_Shutter : Bool;   // Pneu to Machining
      Conveyor1_Sensor : Bool;   // Pneu to Machining
      Cobot_Moving : Bool;   // Pneu to Machining
      Pneumatic_EmergencyBTN : Bool;   // Pneu to Machining
      SetCognexID : Bool;   // Pneu to Machining
      M_PlantView : Bool;   // Pneu to Machining
      M_ManualControl : Bool;   // Pneu to Machining
      M_ProcessTimes : Bool;   // Pneu to Machining
      HMI_BTN_Enter : Bool;   // Pneu to Machining
      HMI_BTN_Logout : Bool;   // Pneu to Machining
      PneumaticPower : Real;   // Pneu to Machining
      AirPressure : Real;   // Pneu to Machining
      ActiveUser : String[40];   // Pneu to Machining
      ActiveRole : String[30];   // Pneu to Machining
      ChocolateCount : Int;   // Pneu to Machining
      VanillaCount : Int;   // Pneu to Machining
      StrawberryCount : Int;   // Pneu to Machining
   END_VAR
BEGIN
END_DATA_BLOCK

// folder: System blocks/Program resources

DATA_BLOCK "TON_Start"   // DB1
{ S7_Optimized_Access := 'TRUE' }
AUTHOR : Simatic
FAMILY : IEC
NAME : IEC_TMR
VERSION : 1.0
// stored: InstanceOfName IEC_TIMER
"IEC_TIMER"
BEGIN
END_DATA_BLOCK

DATA_BLOCK "TOF_Start"   // DB2
{ S7_Optimized_Access := 'TRUE' }
AUTHOR : Simatic
FAMILY : IEC
NAME : IEC_TMR
VERSION : 1.0
// stored: InstanceOfName IEC_TIMER
"IEC_TIMER"
BEGIN
END_DATA_BLOCK

DATA_BLOCK "TON_vertical_piston"   // DB4
{ S7_Optimized_Access := 'TRUE' }
AUTHOR : Simatic
FAMILY : IEC
NAME : IEC_TMR
VERSION : 1.0
// stored: InstanceOfName IEC_TIMER
"IEC_TIMER"
BEGIN
END_DATA_BLOCK

DATA_BLOCK "TON_Turntable"   // DB5
{ S7_Optimized_Access := 'TRUE' }
AUTHOR : Simatic
FAMILY : IEC
NAME : IEC_TMR
VERSION : 1.0
// stored: InstanceOfName IEC_TIMER
"IEC_TIMER"
BEGIN
END_DATA_BLOCK

DATA_BLOCK "TP_piston_in_conveyor"   // DB6
{ S7_Optimized_Access := 'TRUE' }
AUTHOR : Simatic
FAMILY : IEC
NAME : IEC_TMR
VERSION : 1.0
// stored: InstanceOfName IEC_TIMER
"IEC_TIMER"
BEGIN
END_DATA_BLOCK

DATA_BLOCK "TP_ReceiveCognexID"   // DB8
{ S7_Optimized_Access := 'TRUE' }
AUTHOR : Simatic
FAMILY : IEC
NAME : IEC_TMR
VERSION : 1.0
// stored: InstanceOfName IEC_TIMER
"IEC_TIMER"
BEGIN
END_DATA_BLOCK

DATA_BLOCK "TONR_SinceCamScan"   // DB9
{ S7_Optimized_Access := 'TRUE' }
AUTHOR : Simatic
FAMILY : IEC
NAME : IEC_TMR
VERSION : 1.0
// stored: InstanceOfName IEC_TIMER
"IEC_TIMER"
BEGIN
END_DATA_BLOCK

DATA_BLOCK "SetCognexID_TP"   // DB10
{ S7_Optimized_Access := 'TRUE' }
AUTHOR : Simatic
FAMILY : IEC
NAME : IEC_TMR
VERSION : 1.0
// stored: InstanceOfName IEC_TIMER
"IEC_TIMER"
BEGIN
END_DATA_BLOCK

DATA_BLOCK "RelayReceive_TON"   // DB12
{ S7_Optimized_Access := 'TRUE' }
AUTHOR : Simatic
FAMILY : IEC
NAME : IEC_TMR
VERSION : 1.0
// stored: InstanceOfName IEC_TIMER
"IEC_TIMER"
BEGIN
END_DATA_BLOCK

DATA_BLOCK "HMI_Enter_Delay"   // DB14
{ S7_Optimized_Access := 'TRUE' }
AUTHOR : Simatic
FAMILY : IEC
NAME : IEC_TMR
VERSION : 1.0
// stored: InstanceOfName IEC_TIMER
"IEC_TIMER"
BEGIN
END_DATA_BLOCK

DATA_BLOCK "conveyor6_Finish_TP"   // DB15
{ S7_Optimized_Access := 'TRUE' }
AUTHOR : Simatic
FAMILY : IEC
NAME : IEC_TMR
VERSION : 1.0
// stored: InstanceOfName IEC_TIMER
"IEC_TIMER"
BEGIN
END_DATA_BLOCK

DATA_BLOCK "ReceivedCobotByte_TON"   // DB16
{ S7_Optimized_Access := 'TRUE' }
AUTHOR : Simatic
FAMILY : IEC
NAME : IEC_TMR
VERSION : 1.0
// stored: InstanceOfName IEC_TIMER
"IEC_TIMER"
BEGIN
END_DATA_BLOCK

DATA_BLOCK "Chocolate_Counter"   // DB17
{ S7_Optimized_Access := 'TRUE' }
AUTHOR : Simatic
FAMILY : IEC
NAME : CNTR
VERSION : 1.0
// stored: InstanceOfName IEC_COUNTER
"IEC_COUNTER"
BEGIN
END_DATA_BLOCK

DATA_BLOCK "Vanilla_Counter"   // DB18
{ S7_Optimized_Access := 'TRUE' }
AUTHOR : Simatic
FAMILY : IEC
NAME : CNTR
VERSION : 1.0
// stored: InstanceOfName IEC_COUNTER
"IEC_COUNTER"
BEGIN
END_DATA_BLOCK

DATA_BLOCK "Strawberry_Counter"   // DB19
{ S7_Optimized_Access := 'TRUE' }
AUTHOR : Simatic
FAMILY : IEC
NAME : CNTR
VERSION : 1.0
// stored: InstanceOfName IEC_COUNTER
"IEC_COUNTER"
BEGIN
END_DATA_BLOCK

DATA_BLOCK "LogoutBTN_TP"   // DB21
{ S7_Optimized_Access := 'TRUE' }
AUTHOR : Simatic
FAMILY : IEC
NAME : IEC_TMR
VERSION : 1.0
// stored: InstanceOfName IEC_TIMER
"IEC_TIMER"
BEGIN
END_DATA_BLOCK

DATA_BLOCK "CycleTime_TON"   // DB22
{ S7_Optimized_Access := 'TRUE' }
AUTHOR : Simatic
FAMILY : IEC
NAME : IEC_TMR
VERSION : 1.0
// stored: InstanceOfName IEC_TIMER
"IEC_TIMER"
BEGIN
END_DATA_BLOCK

// folder: (top level)

ORGANIZATION_BLOCK "Main_Pneumatic"   // OB1, LAD, ProgramCycle
{ S7_Optimized_Access := 'TRUE' }
VERSION : 0.1
   VAR_INPUT
      Initial_Call : Bool;
      Remanence : Bool;
   END_VAR
   VAR_TEMP   // added for the SCL form of the ladder/FBD networks
      _w1 : Bool;
   END_VAR
BEGIN

REGION Network 1: PUT and GET communication between both PLC's
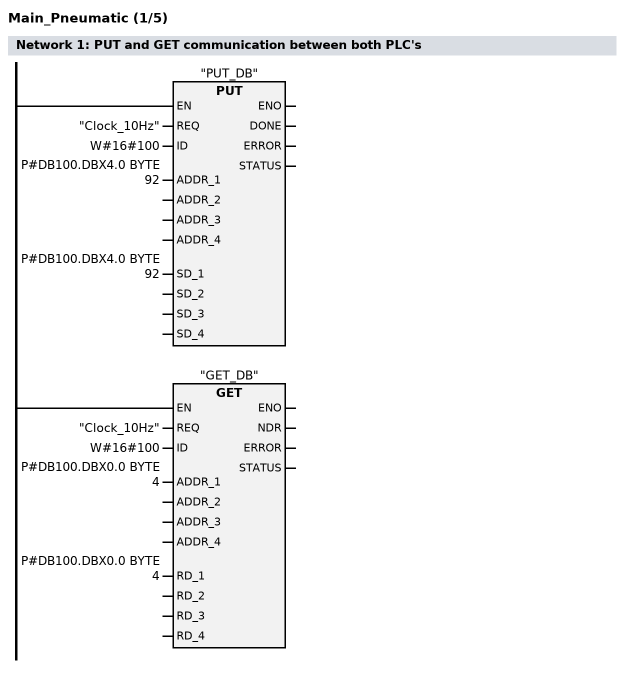
   "PUT_DB"(REQ := "Clock_10Hz",   // PUT
            ID := W#16#100,
            ADDR_1 := P#DB100.DBX4.0 BYTE 92,
            SD_1 := P#DB100.DBX4.0 BYTE 92);
   "GET_DB"(REQ := "Clock_10Hz", ID := W#16#100, ADDR_1 := P#DB100.DBX0.0 BYTE 4, RD_1 := P#DB100.DBX0.0 BYTE 4);   // GET
END_REGION

REGION Network 2: Read Cognex code
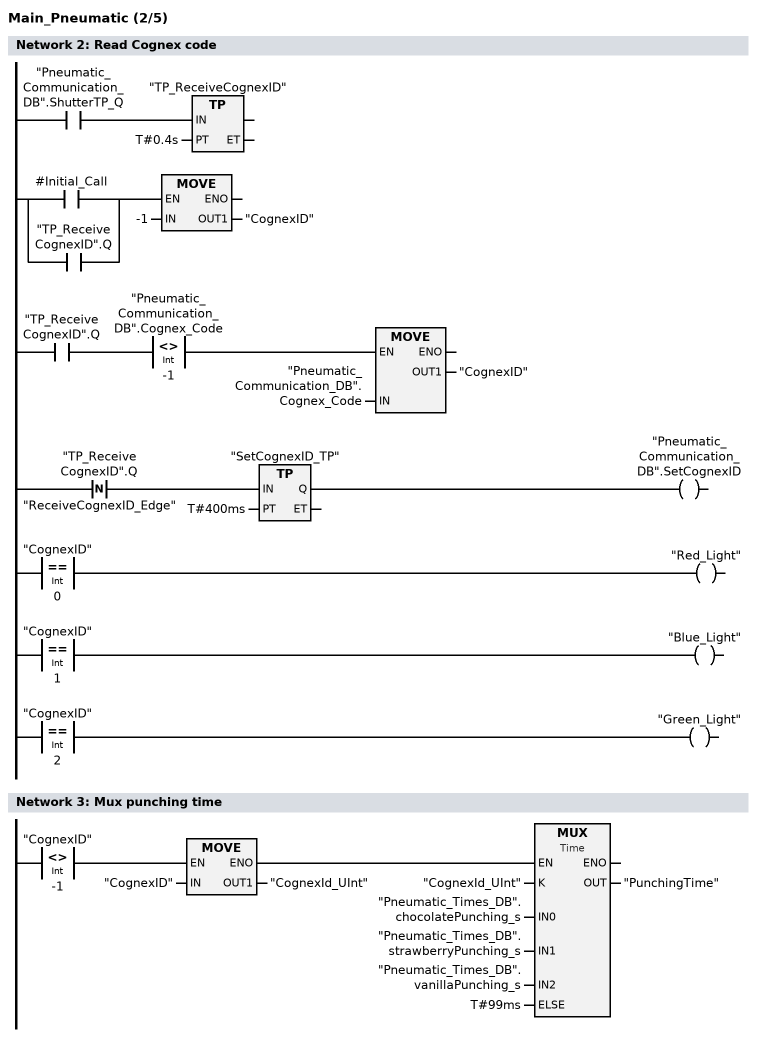
   "TP_ReceiveCognexID".TP(IN := "Pneumatic_Communication_DB".ShutterTP_Q, PT := T#0.4s);
   IF #Initial_Call OR "TP_ReceiveCognexID".Q THEN "CognexID" := -1; END_IF;
   IF "TP_ReceiveCognexID".Q AND ("Pneumatic_Communication_DB".Cognex_Code <> (-1)) THEN
       "CognexID" := "Pneumatic_Communication_DB".Cognex_Code;
   END_IF;
   #_w1 := NOT "TP_ReceiveCognexID".Q AND "ReceiveCognexID_Edge";   // falling edge of "TP_ReceiveCognexID".Q
   "ReceiveCognexID_Edge" := "TP_ReceiveCognexID".Q;
   "SetCognexID_TP".TP(IN := #_w1, PT := T#400ms);
   "Pneumatic_Communication_DB".SetCognexID := "SetCognexID_TP".Q;
   "Red_Light" := "CognexID" = 0;
   "Blue_Light" := "CognexID" = 1;
   "Green_Light" := "CognexID" = 2;
END_REGION

REGION Network 3: Mux punching time
   RUNG wire#powerrail
      { S7_Templates := "SrcType := Int" } NE_Contact(in1 := "CognexID", in2 := -1)
      Move(in := "CognexID", out1 => "CognexId_UInt")
      { S7_Templates := "SrcType := Time"; S7_GenerateENO := "TRUE" } Mux(k := "CognexId_UInt", in0 := "Pneumatic_Times_DB".chocolatePunching_s, in1 := "Pneumatic_Times_DB".strawberryPunching_s, in2 := "Pneumatic_Times_DB".vanillaPunching_s, "else" := T#99ms, out => "PunchingTime")
   END_RUNG
   // the same network as SCL:
   // no SCL statement known for Mux: written as a call
   IF "CognexID" <> (-1) THEN
       "CognexId_UInt" := "CognexID";
       Mux(k := "CognexId_UInt",
           in0 := "Pneumatic_Times_DB".chocolatePunching_s,
           in1 := "Pneumatic_Times_DB".strawberryPunching_s,
           in2 := "Pneumatic_Times_DB".vanillaPunching_s,
           "else" := T#99ms,
           out => "PunchingTime");
   END_IF;
END_REGION

REGION Network 4: Start Piston
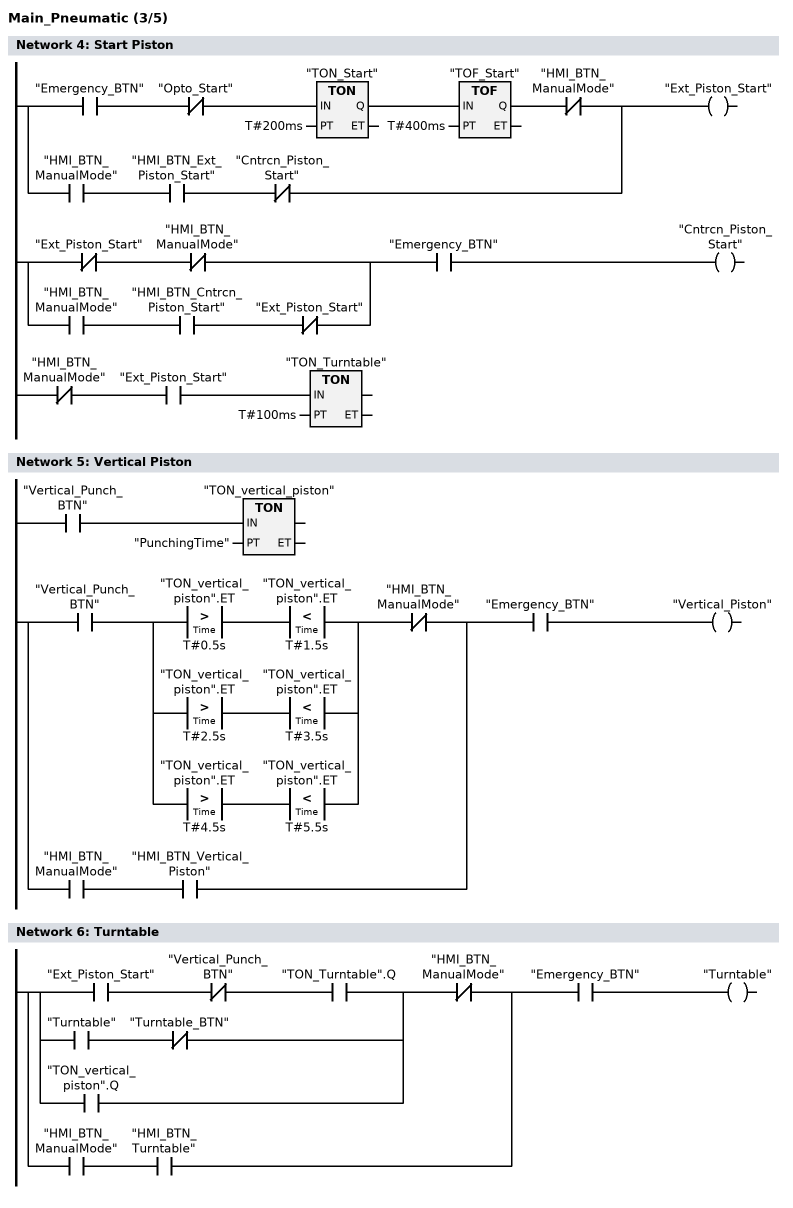
   "TON_Start".TON(IN := "Emergency_BTN" AND NOT "Opto_Start", PT := T#200ms);
   "TOF_Start".TOF(IN := "TON_Start".Q, PT := T#400ms);
   "Ext_Piston_Start" := ("TOF_Start".Q AND NOT "HMI_BTN_ManualMode") OR ("HMI_BTN_ManualMode" AND "HMI_BTN_Ext_Piston_Start" AND NOT "Cntrcn_Piston_Start");
   "Cntrcn_Piston_Start" := ((NOT "Ext_Piston_Start" AND NOT "HMI_BTN_ManualMode") OR ("HMI_BTN_ManualMode" AND "HMI_BTN_Cntrcn_Piston_Start" AND NOT "Ext_Piston_Start")) AND "Emergency_BTN";
   "TON_Turntable".TON(IN := NOT "HMI_BTN_ManualMode" AND "Ext_Piston_Start", PT := T#100ms);
END_REGION

REGION Network 5: Vertical Piston
   "TON_vertical_piston".TON(IN := "Vertical_Punch_BTN", PT := "PunchingTime");
   "Vertical_Piston" := (("Vertical_Punch_BTN" AND ((("TON_vertical_piston".ET > T#0.5s) AND ("TON_vertical_piston".ET < T#1.5s)) OR (("TON_vertical_piston".ET > T#2.5s) AND ("TON_vertical_piston".ET < T#3.5s)) OR (("TON_vertical_piston".ET > T#4.5s) AND ("TON_vertical_piston".ET < T#5.5s))) AND NOT "HMI_BTN_ManualMode") OR ("HMI_BTN_ManualMode" AND "HMI_BTN_Vertical_Piston")) AND "Emergency_BTN";
END_REGION

REGION Network 6: Turntable
   RUNG wire#powerrail
      Contact( "Ext_Piston_Start" )
      I_Contact( "Vertical_Punch_BTN" )
      Contact( "TON_Turntable".Q )
      wire#w1
      I_Contact( "HMI_BTN_ManualMode" )
      wire#w2
      Contact( "Emergency_BTN" )
      Coil( "Turntable" )
   END_RUNG
   RUNG wire#powerrail
      Contact( "Turntable" )
      I_Contact( "Turntable_BTN" )
   END_RUNG wire#w1
   RUNG wire#powerrail
      Contact( "TON_vertical_piston".Q )
   END_RUNG wire#w1
   RUNG wire#powerrail
      Contact( "HMI_BTN_ManualMode" )
      Contact( "HMI_BTN_Turntable" )
   END_RUNG wire#w2
   // the same network as SCL:
   "Turntable" := (((("Ext_Piston_Start" AND NOT "Vertical_Punch_BTN" AND "TON_Turntable".Q) OR ("Turntable" AND NOT "Turntable_BTN") OR "TON_vertical_piston".Q) AND NOT "HMI_BTN_ManualMode") OR ("HMI_BTN_ManualMode" AND "HMI_BTN_Turntable")) AND "Emergency_BTN";
END_REGION

REGION Network 7: Conveyor Piston
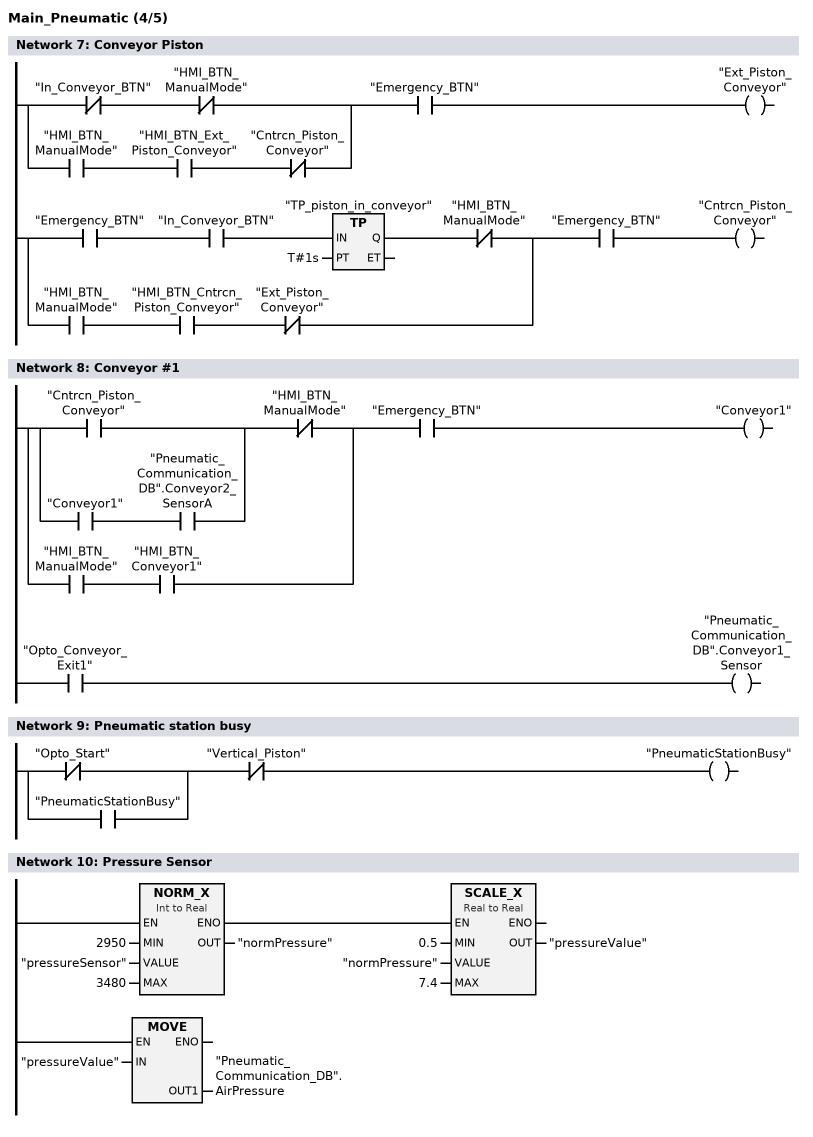
   "Ext_Piston_Conveyor" := ((NOT "In_Conveyor_BTN" AND NOT "HMI_BTN_ManualMode") OR ("HMI_BTN_ManualMode" AND "HMI_BTN_Ext_Piston_Conveyor" AND NOT "Cntrcn_Piston_Conveyor")) AND "Emergency_BTN";
   "TP_piston_in_conveyor".TP(IN := "Emergency_BTN" AND "In_Conveyor_BTN", PT := T#1s);
   "Cntrcn_Piston_Conveyor" := (("TP_piston_in_conveyor".Q AND NOT "HMI_BTN_ManualMode") OR ("HMI_BTN_ManualMode" AND "HMI_BTN_Cntrcn_Piston_Conveyor" AND NOT "Ext_Piston_Conveyor")) AND "Emergency_BTN";
END_REGION

REGION Network 8: Conveyor #1
   RUNG wire#powerrail
      Contact( "Cntrcn_Piston_Conveyor" )
      wire#w1
      I_Contact( "HMI_BTN_ManualMode" )
      wire#w2
      Contact( "Emergency_BTN" )
      Coil( "Conveyor1" )
   END_RUNG
   RUNG wire#powerrail
      Contact( "Conveyor1" )
      Contact( "Pneumatic_Communication_DB".Conveyor2_SensorA )
   END_RUNG wire#w1
   RUNG wire#powerrail
      Contact( "HMI_BTN_ManualMode" )
      Contact( "HMI_BTN_Conveyor1" )
   END_RUNG wire#w2
   RUNG wire#powerrail
      Contact( "Opto_Conveyor_Exit1" )
      Coil( "Pneumatic_Communication_DB".Conveyor1_Sensor )
   END_RUNG
   // the same network as SCL:
   "Conveyor1" := ((("Cntrcn_Piston_Conveyor" OR ("Conveyor1" AND "Pneumatic_Communication_DB".Conveyor2_SensorA)) AND NOT "HMI_BTN_ManualMode") OR ("HMI_BTN_ManualMode" AND "HMI_BTN_Conveyor1")) AND "Emergency_BTN";
   "Pneumatic_Communication_DB".Conveyor1_Sensor := "Opto_Conveyor_Exit1";
END_REGION

REGION Network 9: Pneumatic station busy
   RUNG wire#powerrail
      I_Contact( "Opto_Start" )
      wire#w1
      I_Contact( "Vertical_Piston" )
      Coil( "PneumaticStationBusy" )
   END_RUNG
   RUNG wire#powerrail
      Contact( "PneumaticStationBusy" )
   END_RUNG wire#w1
   // the same network as SCL:
   "PneumaticStationBusy" := (NOT "Opto_Start" OR "PneumaticStationBusy") AND NOT "Vertical_Piston";
END_REGION

REGION Network 10: Pressure Sensor
   RUNG wire#powerrail
      { S7_Templates := "[SrcType := Int, DestType := Real]" } Normalize(min := 2950, value := "pressureSensor", max := 3480, out => "normPressure")
      { S7_Templates := "[SrcType := Real, DestType := Real]" } Scale(min := 0.5, value := "normPressure", max := 7.4, out => "pressureValue")
   END_RUNG
   RUNG wire#powerrail
      Move(in := "pressureValue", out1 => "Pneumatic_Communication_DB".AirPressure)
   END_RUNG
   // the same network as SCL:
   "normPressure" := NORM_X(MIN := 2950, VALUE := "pressureSensor", MAX := 3480);
   "pressureValue" := SCALE_X(MIN := 0.5, VALUE := "normPressure", MAX := 7.4);
   "Pneumatic_Communication_DB".AirPressure := "pressureValue";
END_REGION

REGION Network 11: Initial Photo and time since last photo
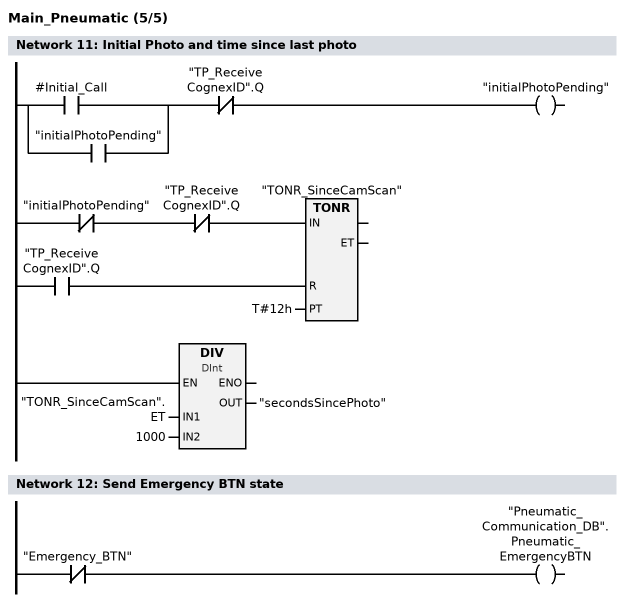
   "initialPhotoPending" := (#Initial_Call OR "initialPhotoPending") AND NOT "TP_ReceiveCognexID".Q;
   "TONR_SinceCamScan".TONR(IN := NOT "initialPhotoPending" AND NOT "TP_ReceiveCognexID".Q,
                           R := "TP_ReceiveCognexID".Q,
                           PT := T#12h);
   "secondsSincePhoto" := "TONR_SinceCamScan".ET / 1000;
END_REGION

REGION Network 12: Send Emergency BTN state
   RUNG wire#powerrail
      I_Contact( "Emergency_BTN" )
      Coil( "Pneumatic_Communication_DB".Pneumatic_EmergencyBTN )
   END_RUNG
   // the same network as SCL:
   "Pneumatic_Communication_DB".Pneumatic_EmergencyBTN := NOT "Emergency_BTN";
END_REGION
END_ORGANIZATION_BLOCK

ORGANIZATION_BLOCK "HMI_OB"   // OB123, LAD, ProgramCycle
{ S7_Optimized_Access := 'TRUE' }
VERSION : 0.1
   VAR_INPUT
      Initial_Call : Bool;
      Remanence : Bool;
   END_VAR
   VAR_TEMP   // added for the SCL form of the ladder/FBD networks
      _w1 : Bool;
   END_VAR
BEGIN

REGION Network 1: Set HMI screen to 0 (acces Screen) on startup
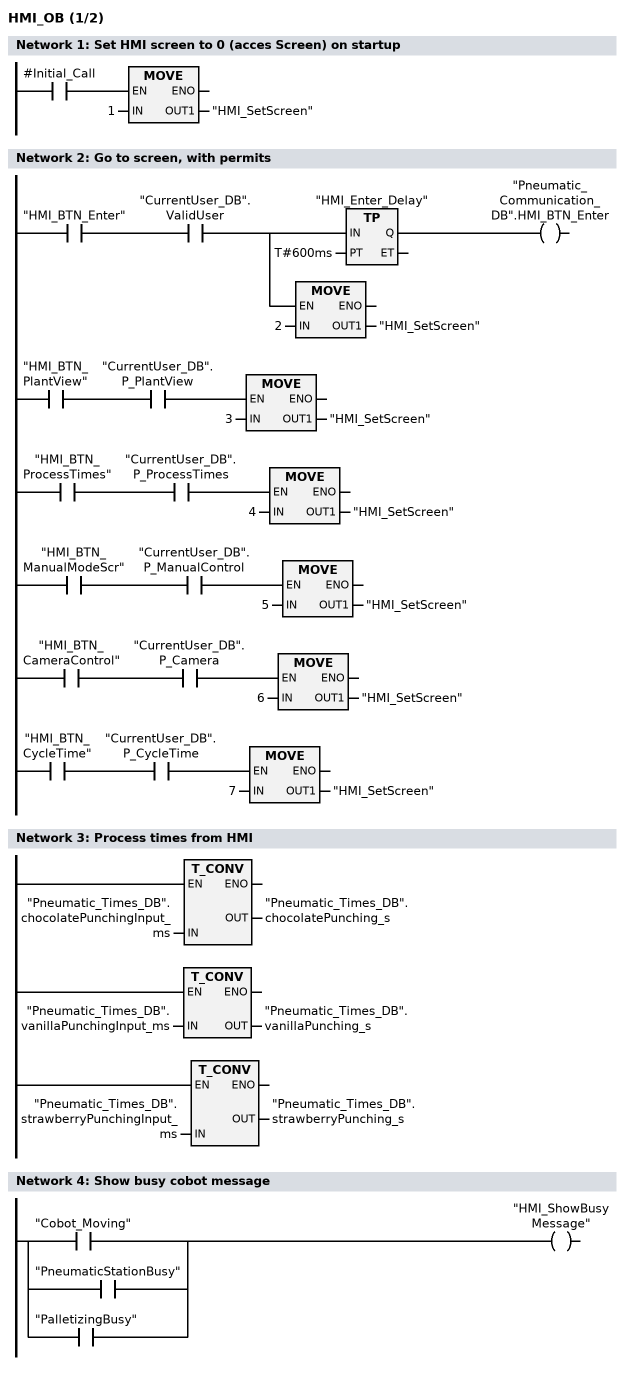
   RUNG wire#powerrail
      Contact( #Initial_Call )
      Move(in := 1, out1 => "HMI_SetScreen")
   END_RUNG
   // the same network as SCL:
   IF #Initial_Call THEN "HMI_SetScreen" := 1; END_IF;
END_REGION

REGION Network 2: Go to screen, with permits
   #_w1 := "HMI_BTN_Enter" AND "CurrentUser_DB".ValidUser;
   "HMI_Enter_Delay".TP(IN := #_w1, PT := T#600ms);
   "Pneumatic_Communication_DB".HMI_BTN_Enter := "HMI_Enter_Delay".Q;
   IF #_w1 THEN "HMI_SetScreen" := 2; END_IF;
   IF "HMI_BTN_PlantView" AND "CurrentUser_DB".P_PlantView THEN "HMI_SetScreen" := 3; END_IF;
   IF "HMI_BTN_ProcessTimes" AND "CurrentUser_DB".P_ProcessTimes THEN "HMI_SetScreen" := 4; END_IF;
   IF "HMI_BTN_ManualModeScr" AND "CurrentUser_DB".P_ManualControl THEN "HMI_SetScreen" := 5; END_IF;
   IF "HMI_BTN_CameraControl" AND "CurrentUser_DB".P_Camera THEN "HMI_SetScreen" := 6; END_IF;
   IF "HMI_BTN_CycleTime" AND "CurrentUser_DB".P_CycleTime THEN "HMI_SetScreen" := 7; END_IF;
END_REGION

REGION Network 3: Process times from HMI
   "Pneumatic_Times_DB".chocolatePunching_s := T_CONV(IN := "Pneumatic_Times_DB".chocolatePunchingInput_ms);
   "Pneumatic_Times_DB".vanillaPunching_s := T_CONV(IN := "Pneumatic_Times_DB".vanillaPunchingInput_ms);
   "Pneumatic_Times_DB".strawberryPunching_s := T_CONV(IN := "Pneumatic_Times_DB".strawberryPunchingInput_ms);
END_REGION

REGION Network 4: Show busy cobot message
   RUNG wire#powerrail
      Contact( "Cobot_Moving" )
      wire#w1
      Coil( "HMI_ShowBusyMessage" )
   END_RUNG
   RUNG wire#powerrail
      Contact( "PneumaticStationBusy" )
   END_RUNG wire#w1
   RUNG wire#powerrail
      Contact( "PalletizingBusy" )
   END_RUNG wire#w1
   // the same network as SCL:
   "HMI_ShowBusyMessage" := "Cobot_Moving" OR "PneumaticStationBusy" OR "PalletizingBusy";
END_REGION

REGION Network 5: Cognex Shutter BTN
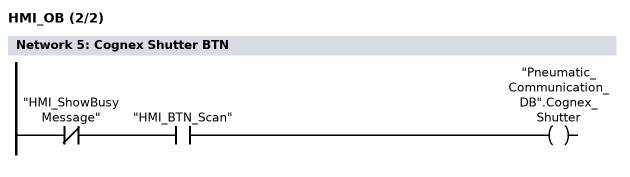
   RUNG wire#powerrail
      I_Contact( "HMI_ShowBusyMessage" )
      Contact( "HMI_BTN_Scan" )
      Coil( "Pneumatic_Communication_DB".Cognex_Shutter )
   END_RUNG
   // the same network as SCL:
   "Pneumatic_Communication_DB".Cognex_Shutter := NOT "HMI_ShowBusyMessage" AND "HMI_BTN_Scan";
END_REGION
END_ORGANIZATION_BLOCK

ORGANIZATION_BLOCK "Cobot_OB"   // OB124, LAD, ProgramCycle
{ S7_Optimized_Access := 'TRUE' }
VERSION : 0.1
   VAR_INPUT
      Initial_Call : Bool;
      Remanence : Bool;
   END_VAR
BEGIN

REGION Network 1: Read cobot outputs and form Byte
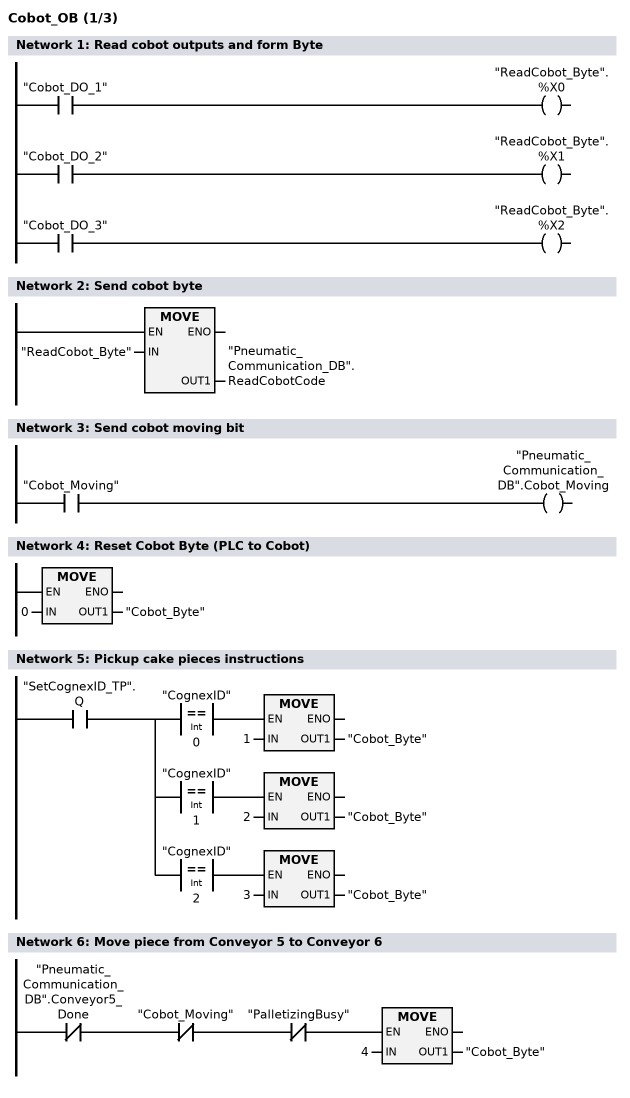
   RUNG wire#powerrail
      Contact( "Cobot_DO_1" )
      Coil( "ReadCobot_Byte".%X0 )
   END_RUNG
   RUNG wire#powerrail
      Contact( "Cobot_DO_2" )
      Coil( "ReadCobot_Byte".%X1 )
   END_RUNG
   RUNG wire#powerrail
      Contact( "Cobot_DO_3" )
      Coil( "ReadCobot_Byte".%X2 )
   END_RUNG
   // the same network as SCL:
   "ReadCobot_Byte".%X0 := "Cobot_DO_1";
   "ReadCobot_Byte".%X1 := "Cobot_DO_2";
   "ReadCobot_Byte".%X2 := "Cobot_DO_3";
END_REGION

REGION Network 2: Send cobot byte
   RUNG wire#powerrail
      Move(in := "ReadCobot_Byte", out1 => "Pneumatic_Communication_DB".ReadCobotCode)
   END_RUNG
   // the same network as SCL:
   "Pneumatic_Communication_DB".ReadCobotCode := "ReadCobot_Byte";
END_REGION

REGION Network 3: Send cobot moving bit
   RUNG wire#powerrail
      Contact( "Cobot_Moving" )
      Coil( "Pneumatic_Communication_DB".Cobot_Moving )
   END_RUNG
   // the same network as SCL:
   "Pneumatic_Communication_DB".Cobot_Moving := "Cobot_Moving";
END_REGION

REGION Network 4: Reset Cobot Byte (PLC to Cobot)
   RUNG wire#powerrail
      Move(in := 0, out1 => "Cobot_Byte")
   END_RUNG
   // the same network as SCL:
   "Cobot_Byte" := 0;
END_REGION

REGION Network 5: Pickup cake pieces instructions
   RUNG wire#powerrail
      Contact( "SetCognexID_TP".Q )
      wire#w1
      { S7_Templates := "SrcType := Int" } EQ_Contact(in1 := "CognexID", in2 := 0)
      Move(in := 1, out1 => "Cobot_Byte")
   END_RUNG
   RUNG wire#w1
      { S7_Templates := "SrcType := Int" } EQ_Contact(in1 := "CognexID", in2 := 1)
      Move(in := 2, out1 => "Cobot_Byte")
   END_RUNG
   RUNG wire#w1
      { S7_Templates := "SrcType := Int" } EQ_Contact(in1 := "CognexID", in2 := 2)
      Move(in := 3, out1 => "Cobot_Byte")
   END_RUNG
   // the same network as SCL:
   IF "SetCognexID_TP".Q AND ("CognexID" = 0) THEN "Cobot_Byte" := 1; END_IF;
   IF "SetCognexID_TP".Q AND ("CognexID" = 1) THEN "Cobot_Byte" := 2; END_IF;
   IF "SetCognexID_TP".Q AND ("CognexID" = 2) THEN "Cobot_Byte" := 3; END_IF;
END_REGION

REGION Network 6: Move piece from Conveyor 5 to Conveyor 6
   RUNG wire#powerrail
      I_Contact( "Pneumatic_Communication_DB".Conveyor5_Done )
      I_Contact( "Cobot_Moving" )
      I_Contact( "PalletizingBusy" )
      Move(in := 4, out1 => "Cobot_Byte")
   END_RUNG
   // the same network as SCL:
   IF NOT "Pneumatic_Communication_DB".Conveyor5_Done AND NOT "Cobot_Moving" AND NOT "PalletizingBusy" THEN
       "Cobot_Byte" := 4;
   END_IF;
END_REGION

REGION Network 7: Read the palletizing byte for the cobot and set it to the Cobot Byte
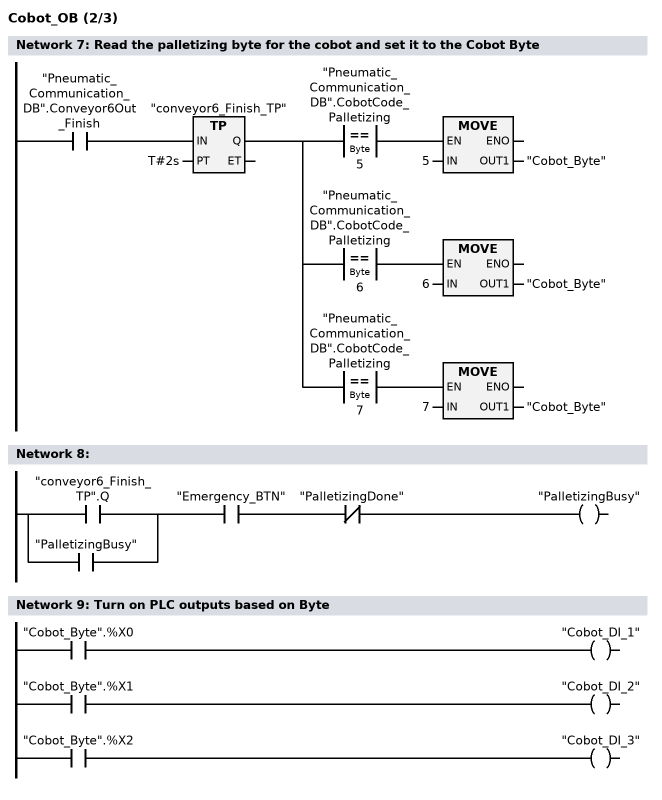
   "conveyor6_Finish_TP".TP(IN := "Pneumatic_Communication_DB".Conveyor6Out_Finish, PT := T#2s);
   IF "conveyor6_Finish_TP".Q AND ("Pneumatic_Communication_DB".CobotCode_Palletizing = 5) THEN
       "Cobot_Byte" := 5;
   END_IF;
   IF "conveyor6_Finish_TP".Q AND ("Pneumatic_Communication_DB".CobotCode_Palletizing = 6) THEN
       "Cobot_Byte" := 6;
   END_IF;
   IF "conveyor6_Finish_TP".Q AND ("Pneumatic_Communication_DB".CobotCode_Palletizing = 7) THEN
       "Cobot_Byte" := 7;
   END_IF;
END_REGION

REGION Network 8
   RUNG wire#powerrail
      Contact( "conveyor6_Finish_TP".Q )
      wire#w1
      Contact( "Emergency_BTN" )
      I_Contact( "PalletizingDone" )
      Coil( "PalletizingBusy" )
   END_RUNG
   RUNG wire#powerrail
      Contact( "PalletizingBusy" )
   END_RUNG wire#w1
   // the same network as SCL:
   "PalletizingBusy" := ("conveyor6_Finish_TP".Q OR "PalletizingBusy") AND "Emergency_BTN" AND NOT "PalletizingDone";
END_REGION

REGION Network 9: Turn on PLC outputs based on Byte
   RUNG wire#powerrail
      Contact( "Cobot_Byte".%X0 )
      Coil( "Cobot_DI_1" )
   END_RUNG
   RUNG wire#powerrail
      Contact( "Cobot_Byte".%X1 )
      Coil( "Cobot_DI_2" )
   END_RUNG
   RUNG wire#powerrail
      Contact( "Cobot_Byte".%X2 )
      Coil( "Cobot_DI_3" )
   END_RUNG
   // the same network as SCL:
   "Cobot_DI_1" := "Cobot_Byte".%X0;
   "Cobot_DI_2" := "Cobot_Byte".%X1;
   "Cobot_DI_3" := "Cobot_Byte".%X2;
END_REGION

REGION Network 10: Produced pieces counter
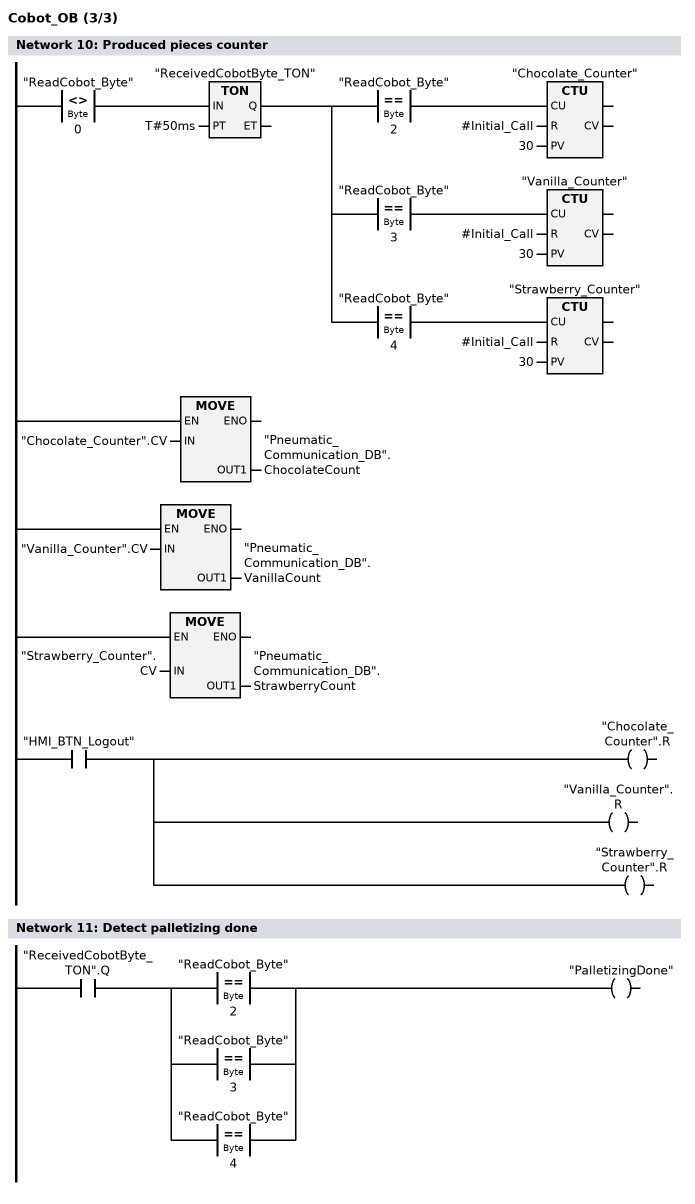
   "ReceivedCobotByte_TON".TON(IN := "ReadCobot_Byte" <> 0, PT := T#50ms);
   "Chocolate_Counter".CTU(CU := "ReceivedCobotByte_TON".Q AND ("ReadCobot_Byte" = 2),
                           R := #Initial_Call,
                           PV := 30);
   "Vanilla_Counter".CTU(CU := "ReceivedCobotByte_TON".Q AND ("ReadCobot_Byte" = 3),
                         R := #Initial_Call,
                         PV := 30);
   "Strawberry_Counter".CTU(CU := "ReceivedCobotByte_TON".Q AND ("ReadCobot_Byte" = 4),
                           R := #Initial_Call,
                           PV := 30);
   "Pneumatic_Communication_DB".ChocolateCount := "Chocolate_Counter".CV;
   "Pneumatic_Communication_DB".VanillaCount := "Vanilla_Counter".CV;
   "Pneumatic_Communication_DB".StrawberryCount := "Strawberry_Counter".CV;
   "Chocolate_Counter".R := "HMI_BTN_Logout";
   "Vanilla_Counter".R := "HMI_BTN_Logout";
   "Strawberry_Counter".R := "HMI_BTN_Logout";
END_REGION

REGION Network 11: Detect palletizing done
   RUNG wire#powerrail
      Contact( "ReceivedCobotByte_TON".Q )
      wire#w1
      { S7_Templates := "SrcType := Byte" } EQ_Contact(in1 := "ReadCobot_Byte", in2 := 2)
      wire#w2
      Coil( "PalletizingDone" )
   END_RUNG
   RUNG wire#w1
      { S7_Templates := "SrcType := Byte" } EQ_Contact(in1 := "ReadCobot_Byte", in2 := 3)
   END_RUNG wire#w2
   RUNG wire#w1
      { S7_Templates := "SrcType := Byte" } EQ_Contact(in1 := "ReadCobot_Byte", in2 := 4)
   END_RUNG wire#w2
   // the same network as SCL:
   "PalletizingDone" := "ReceivedCobotByte_TON".Q AND (("ReadCobot_Byte" = 2) OR ("ReadCobot_Byte" = 3) OR ("ReadCobot_Byte" = 4));
END_REGION
END_ORGANIZATION_BLOCK

ORGANIZATION_BLOCK "MonitoringPneumatic_OB"   // OB125, LAD, ProgramCycle
{ S7_Optimized_Access := 'TRUE' }
VERSION : 0.1
   VAR_INPUT
      Initial_Call : Bool;
      Remanence : Bool;
   END_VAR
BEGIN

REGION Network 1: Monitor Power consumption (W)
